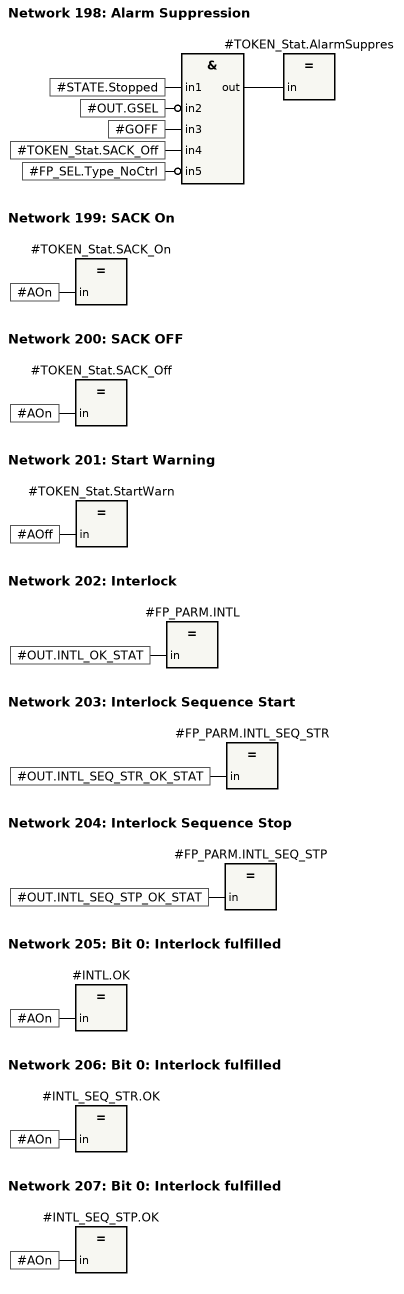
   #TOKEN_Stat.AlarmSuppres := #STATE.Stopped AND NOT #OUT.GSEL AND #GOFF AND #TOKEN_Stat.SACK_Off AND NOT #FP_SEL.Type_NoCtrl;
END_REGION

REGION Network 199: SACK On
   #TOKEN_Stat.SACK_On := #AOn;
END_REGION

REGION Network 200: SACK OFF
   #TOKEN_Stat.SACK_Off := #AOn;
END_REGION

REGION Network 201: Start Warning
   #TOKEN_Stat.StartWarn := #AOff;
END_REGION

REGION Network 202: Interlock
   #FP_PARM.INTL := #OUT.INTL_OK_STAT;
END_REGION

REGION Network 203: Interlock Sequence Start
   #FP_PARM.INTL_SEQ_STR := #OUT.INTL_SEQ_STR_OK_STAT;
END_REGION

REGION Network 204: Interlock Sequence Stop
   #FP_PARM.INTL_SEQ_STP := #OUT.INTL_SEQ_STP_OK_STAT;
END_REGION

REGION Network 205: Bit 0: Interlock fulfilled
   #INTL.OK := #AOn;
END_REGION

REGION Network 206: Bit 0: Interlock fulfilled
   #INTL_SEQ_STR.OK := #AOn;
END_REGION

REGION Network 207: Bit 0: Interlock fulfilled
   #INTL_SEQ_STP.OK := #AOn;
END_REGION

REGION Network 208: Bit 1: Detect first occuring interlock, unit running
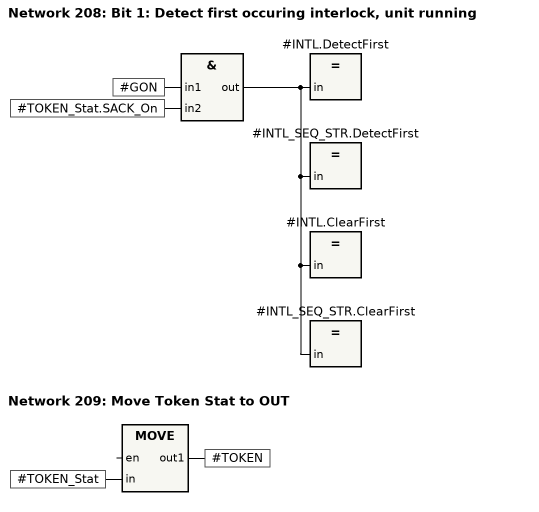
   #INTL.DetectFirst := #GON AND #TOKEN_Stat.SACK_On;
   #INTL_SEQ_STR.DetectFirst := #INTL.DetectFirst;
   #INTL.ClearFirst := #INTL.DetectFirst;
   #INTL_SEQ_STR.ClearFirst := #INTL.DetectFirst;
END_REGION

REGION Network 209: Move Token Stat to OUT
   #TOKEN := #TOKEN_Stat;
END_REGION

REGION Network 210: Write STAT to OUT
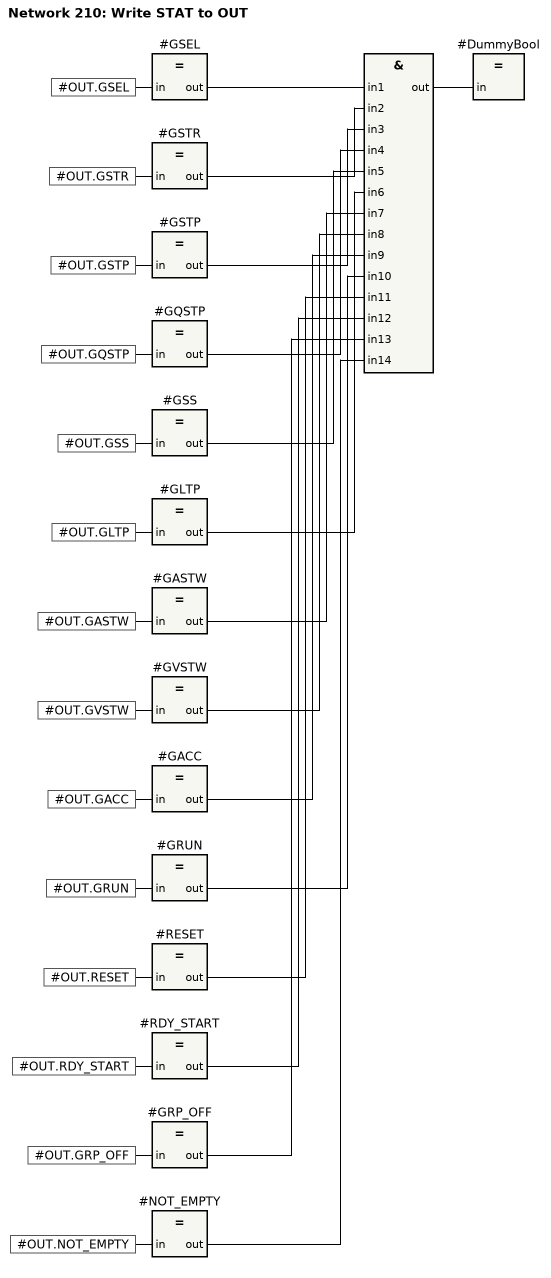
   #GSEL := #OUT.GSEL;
   #GSTR := #OUT.GSTR;
   #GSTP := #OUT.GSTP;
   #GQSTP := #OUT.GQSTP;
   #GSS := #OUT.GSS;
   #GLTP := #OUT.GLTP;
   #GASTW := #OUT.GASTW;
   #GVSTW := #OUT.GVSTW;
   #GACC := #OUT.GACC;
   #GRUN := #OUT.GRUN;
   #RESET := #OUT.RESET;
   #RDY_START := #OUT.RDY_START;
   #GRP_OFF := #OUT.GRP_OFF;
   #NOT_EMPTY := #OUT.NOT_EMPTY;
   #DummyBool := #OUT.GSEL AND #OUT.GSTR AND #OUT.GSTP AND #OUT.GQSTP AND #OUT.GSS AND #OUT.GLTP AND #OUT.GASTW AND #OUT.GVSTW AND #OUT.GACC AND #OUT.GRUN AND #OUT.RESET AND #OUT.RDY_START AND #OUT.GRP_OFF AND #OUT.NOT_EMPTY;
END_REGION
END_FUNCTION_BLOCK

FUNCTION_BLOCK "ACESYS_ALARM"   // FB203, FBD
TITLE = ACESYS V8.0 - Build 004 - Alarm Block
{ S7_Optimized_Access := 'FALSE' }
AUTHOR : FLSmidth
FAMILY : ACESYS
NAME : ALARM
VERSION : 8.0
   VAR_INPUT
      SIG : Bool := TRUE;   // Signal
      PWR : Bool;   // Power Supply
      EN_L : Bool;   // Enable Low Alarm
      EN_H : Bool;   // Enable High Alarm
      AL_SUPR : Bool;   // Alarm Supress by Program
   END_VAR
   VAR_OUTPUT
      OK : Bool;   // Status OK = No Current Alarm
      AL_L : Bool;   // Alarm Low
      AL_H : Bool;   // Alarm High
      WARN_L : Bool;   // Warning Low
      WARN_H : Bool;   // Warning High
      MSW : "ACESYS_HMI_STAT_32T";
   END_VAR
   VAR_IN_OUT
      TOKEN : "ACESYS_TOKEN";
   END_VAR
   VAR
      BlockInfo : Struct
         Ace_Version : Int;   // Acesys Block Version Number
         Ace_BuildNo : Int;   // Acesys Block Build Number
         State_Act : Int;   // Actual State Number
         State_Prev : Int;   // Previous State Number
         DB_Number : Int;   // Block Instance DB Number
      END_STRUCT;
      FP_CMD : Struct   // Faceplate Commands
         Spare_08 : Bool;
         Spare_09 : Bool;
         Spare_10 : Bool;
         Spare_11 : Bool;
         Spare_12 : Bool;
         Spare_13 : Bool;
         Spare_14 : Bool;
         AckAlarm : Bool;
         Spare_00 : Bool;
         Spare_01 : Bool;
         Spare_02 : Bool;
         Spare_03 : Bool;
         Spare_04 : Bool;
         Spare_05 : Bool;
         Spare_06 : Bool;
         Spare_07 : Bool;
      END_STRUCT;
      FP_SEL : Struct
         Force_Low_Alarm : Bool;   // Select Bit
         Force_High_Alarm : Bool;   // Select Bit
         Force_OK : Bool;   // Select Bit
         Force_Low_Warning : Bool;   // Select Bit
         Force_High_Warning : Bool;   // Select Bit
         Keep_Status : Bool;   // Select Bit
         Spare06 : Bool;
         Spare07 : Bool;
         Spare08 : Bool;
         Spare09 : Bool;
         Spare10 : Bool;
         Spare11 : Bool;
         Spare12 : Bool;
         Spare13 : Bool;
         Spare14 : Bool;
         Spare15 : Bool;
      END_STRUCT;
      FP_PARM : Struct
         EnableTime_Low_Pre : Int;
         EnableTime_Low_Acc : Int;
         EnableTime_High_Pre : Int;
         EnableTime_High_Acc : Int;
         WarnDelay_Low_Pre : Int;
         WarnDelay_Low_Acc : Int;
         WarnDelay_High_Pre : Int;
         WarnDelay_High_Acc : Int;
         AlarmDelay_High_Pre : Int;
         AlarmDelay_High_Acc : Int;
         AlarmDelay_Low_Pre : Int;
         AlarmDelay_Low_Acc : Int;
         RepeatTime_Pre : Int;
         RepeatTime_Acc : Int;
         Struct0 : Int;
      END_STRUCT;
      FP_EN : Struct
         ParentSupress : Bool;   // Enable Bit
         ParentSupressUnit : Bool;   // Enable Bit
         Repeat_Alarm : Bool;   // Enable Bit
         Alarm_Low : Bool;   // Enable Bit
         Alarm_High : Bool;   // Enable Bit
         Warning_Low : Bool;   // Enable Bit
         Warning_High : Bool;   // Enable Bit
         Spare07 : Bool;
         Spare08 : Bool;
         Spare09 : Bool;
         Spare10 : Bool;
         Spare11 : Bool;
         Spare12 : Bool;
         Spare13 : Bool;
         Spare14 : Bool;
         Spare15 : Bool;
      END_STRUCT;
      FP_SIM : "ACESYS_SIM_ALARM";
      ONS : Struct
         Sec_Pulse2 : Bool;   // OneShot bit
         Sec_Pulse1 : Bool;   // OneShot bit
         Acknowledge : Bool;   // OneShot bit
         ForceOK : Bool;   // OneShot bit
         ForceLowAlarm : Bool;   // OneShot bit
         ForceHighAlarm : Bool;   // OneShot bit
         SecPulse1 : Bool;
         SecPulse2 : Bool;
         Spare08 : Bool;
         Spare07 : Bool;
         Spare06 : Bool;
         Spare05 : Bool;
         Spare04 : Bool;
         ALARM_AlarmCondition : Bool;
         AL_L_Aux : Bool;
         AL_H_Aux : Bool;
      END_STRUCT;
      EnableTime_Low_Done : Bool;   // Timer Done
      EnableTime_High_Done : Bool;   // Timer Done
      WarnDelay_Low_Done : Bool;   // Timer Done
      WarnDelay_High_Done : Bool;   // Timer Done
      AlarmDelay_Low_Done : Bool;   // Timer Done
      AlarmDelay_High_Done : Bool;   // Timer Done
      RepeatTime_Done : Bool;   // Timer Done
      ALARM_SuppresionActiv : Bool;
      ALARM_AlarmPresent : Bool;
      ALARM_WarnPresent : Bool;
      ALARM_Failure_Ack_Requ : Bool;
      ALARM_Warn_Ack_Required : Bool;
      Keep_L_Alarm : Bool;   // Keep Alarm
      Keep_H_Alarm : Bool;
      Sec_Pulse : Bool;   // Pulse Every Second
      CMD_Acknowledge : Bool;   // Internal Acknowledge
      StatusWork : Int;
      AlarmNo : Int;
      AlarmNo_Old : Int;
      EnableTime_Low_Mem : Int;   // Timer Memory
      EnableTime_High_Mem : Int;   // Timer Memory
      WarnDelay_Low_Mem : Int;   // Timer Memory
      WarnDelay_High_Mem : Int;   // Timer Memory
      AlarmDelay_High_Mem : Int;   // Timer Memory
      AlarmDelay_Low_Mem : Int;   // Timer Memory
      RepeatTime_Mem : Int;   // Timer Memory
      OUT : Struct
         OK : Bool;
         AL_L : Bool;
         AL_H : Bool;
         WARN_L : Bool;
         WARN_H : Bool;
      END_STRUCT;
      MSW_EXT_AlarmFailUnAck : Bool;
      MSW_Status_Trans : Int;
   END_VAR
   VAR_TEMP
      AOn : Bool;   // Always On
      AOff : Bool;   // Always Off
      DummyBool : Bool;
   END_VAR
   VAR_TEMP   // added for the SCL form of the ladder/FBD networks
      _w1 : Bool;
      _w2 : Bool;
      _w3 : Bool;
   END_VAR
BEGIN

REGION Network 1: Always On
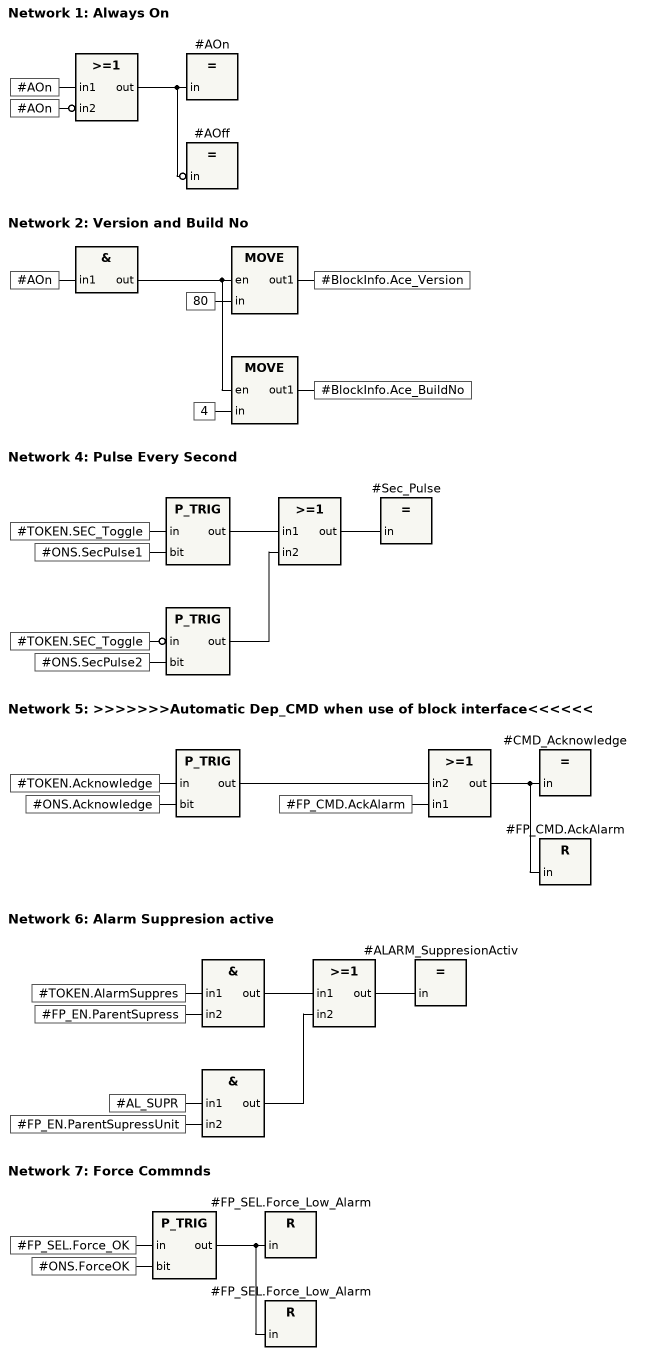
   #AOn := #AOn OR NOT #AOn;
   #AOff := NOT #AOn;
END_REGION

REGION Network 2: Version and Build No
   IF #AOn THEN
       #BlockInfo.Ace_Version := 80;
       #BlockInfo.Ace_BuildNo := 4;
   END_IF;
END_REGION

REGION Network 3 (STL): Instance DB Number to Faceplate
         L     DINO;
         T     #BlockInfo.DB_Number;
END_REGION

REGION Network 4: Pulse Every Second
   #_w1 := #TOKEN.SEC_Toggle AND NOT #ONS.SecPulse1;   // rising edge
   #ONS.SecPulse1 := #TOKEN.SEC_Toggle;
   #_w2 := NOT #TOKEN.SEC_Toggle AND NOT #ONS.SecPulse2;   // rising edge
   #ONS.SecPulse2 := NOT #TOKEN.SEC_Toggle;
   #Sec_Pulse := #_w1 OR #_w2;
END_REGION

REGION Network 5: >>>>>>>Automatic Dep_CMD when use of block interface<<<<<<
   #_w1 := #TOKEN.Acknowledge AND NOT #ONS.Acknowledge;   // rising edge
   #ONS.Acknowledge := #TOKEN.Acknowledge;
   #CMD_Acknowledge := #_w1 OR #FP_CMD.AckAlarm;
   IF #CMD_Acknowledge THEN #FP_CMD.AckAlarm := FALSE; END_IF;
END_REGION

REGION Network 6: Alarm Suppresion active
   #ALARM_SuppresionActiv := (#TOKEN.AlarmSuppres AND #FP_EN.ParentSupress) OR (#AL_SUPR AND #FP_EN.ParentSupressUnit);
END_REGION

REGION Network 7: Force Commnds
   #_w1 := #FP_SEL.Force_OK AND NOT #ONS.ForceOK;   // rising edge
   #ONS.ForceOK := #FP_SEL.Force_OK;
   IF #_w1 THEN
       #FP_SEL.Force_Low_Alarm := FALSE;
       #FP_SEL.Force_Low_Alarm := FALSE;
   END_IF;
END_REGION

REGION Network 8: Select Bit
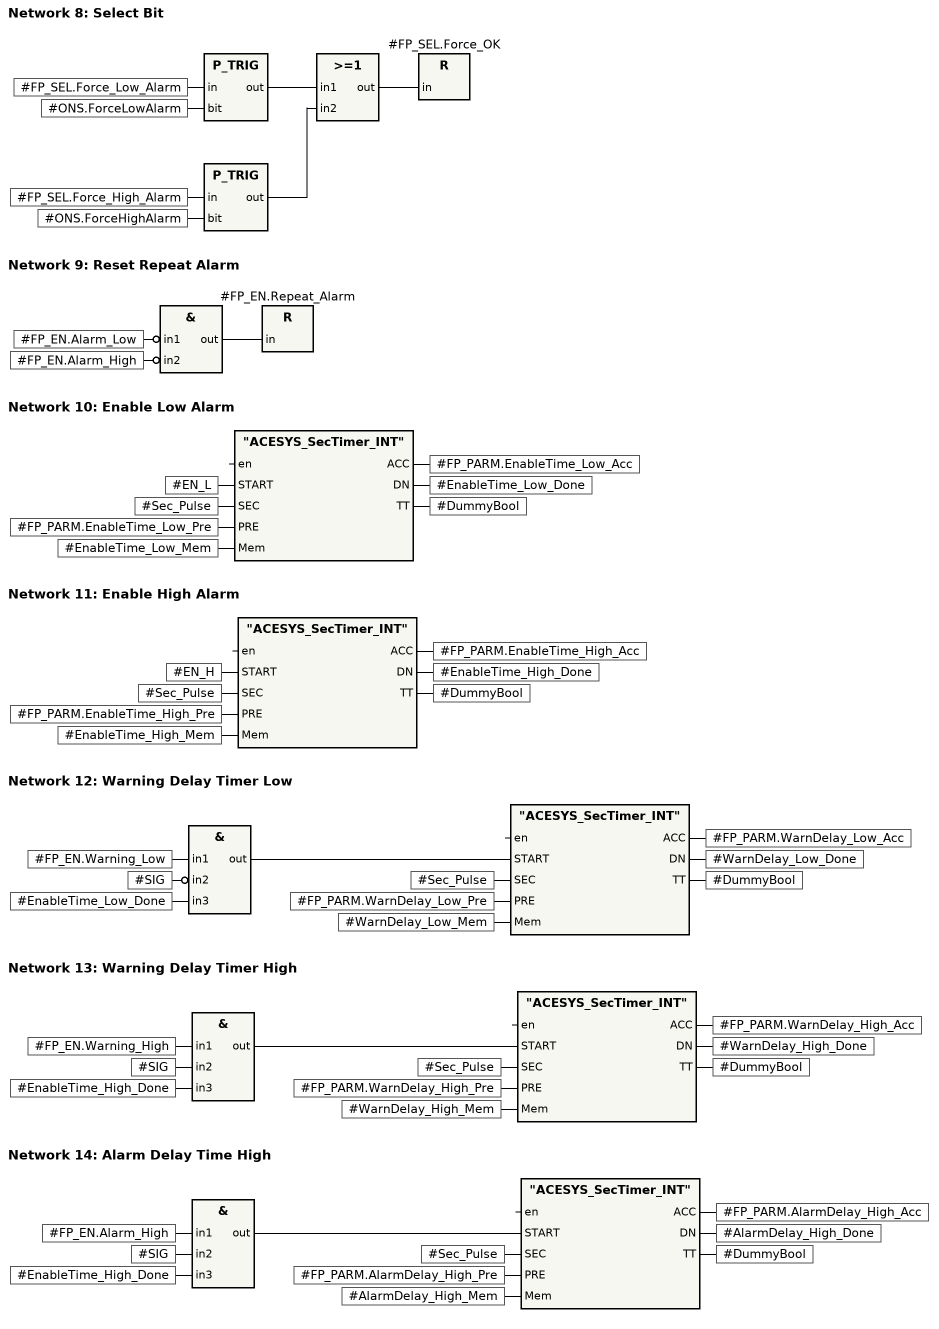
   #_w1 := #FP_SEL.Force_Low_Alarm AND NOT #ONS.ForceLowAlarm;   // rising edge
   #ONS.ForceLowAlarm := #FP_SEL.Force_Low_Alarm;
   #_w2 := #FP_SEL.Force_High_Alarm AND NOT #ONS.ForceHighAlarm;   // rising edge
   #ONS.ForceHighAlarm := #FP_SEL.Force_High_Alarm;
   IF #_w1 OR #_w2 THEN #FP_SEL.Force_OK := FALSE; END_IF;
END_REGION

REGION Network 9: Reset Repeat Alarm
   IF NOT #FP_EN.Alarm_Low AND NOT #FP_EN.Alarm_High THEN #FP_EN.Repeat_Alarm := FALSE; END_IF;
END_REGION

REGION Network 10: Enable Low Alarm
   "ACESYS_SecTimer_INT"(START := #EN_L,
                         SEC := #Sec_Pulse,
                         PRE := #FP_PARM.EnableTime_Low_Pre,
                         Mem := #EnableTime_Low_Mem,
                         ACC => #FP_PARM.EnableTime_Low_Acc,
                         DN => #EnableTime_Low_Done,
                         TT => #DummyBool);
END_REGION

REGION Network 11: Enable High Alarm
   "ACESYS_SecTimer_INT"(START := #EN_H,
                         SEC := #Sec_Pulse,
                         PRE := #FP_PARM.EnableTime_High_Pre,
                         Mem := #EnableTime_High_Mem,
                         ACC => #FP_PARM.EnableTime_High_Acc,
                         DN => #EnableTime_High_Done,
                         TT => #DummyBool);
END_REGION

REGION Network 12: Warning Delay Timer Low
   // Build 002 - 27 March 2019 : EnableTime_Low_Done added
   "ACESYS_SecTimer_INT"(START := #FP_EN.Warning_Low AND NOT #SIG AND #EnableTime_Low_Done,
                         SEC := #Sec_Pulse,
                         PRE := #FP_PARM.WarnDelay_Low_Pre,
                         Mem := #WarnDelay_Low_Mem,
                         ACC => #FP_PARM.WarnDelay_Low_Acc,
                         DN => #WarnDelay_Low_Done,
                         TT => #DummyBool);
END_REGION

REGION Network 13: Warning Delay Timer High
   // Build 002 - 27 March 2019 : EnableTime_High_Done added
   "ACESYS_SecTimer_INT"(START := #FP_EN.Warning_High AND #SIG AND #EnableTime_High_Done,
                         SEC := #Sec_Pulse,
                         PRE := #FP_PARM.WarnDelay_High_Pre,
                         Mem := #WarnDelay_High_Mem,
                         ACC => #FP_PARM.WarnDelay_High_Acc,
                         DN => #WarnDelay_High_Done,
                         TT => #DummyBool);
END_REGION

REGION Network 14: Alarm Delay Time High
   // Build 002 - 27 March 2019 : EnableTime_High_Done added
   "ACESYS_SecTimer_INT"(START := #FP_EN.Alarm_High AND #SIG AND #EnableTime_High_Done,
                         SEC := #Sec_Pulse,
                         PRE := #FP_PARM.AlarmDelay_High_Pre,
                         Mem := #AlarmDelay_High_Mem,
                         ACC => #FP_PARM.AlarmDelay_High_Acc,
                         DN => #AlarmDelay_High_Done,
                         TT => #DummyBool);
END_REGION

REGION Network 15: Alarm Delay Time Low
   // Build 002 - 27 March 2019 : EnableTime_Low_Done added
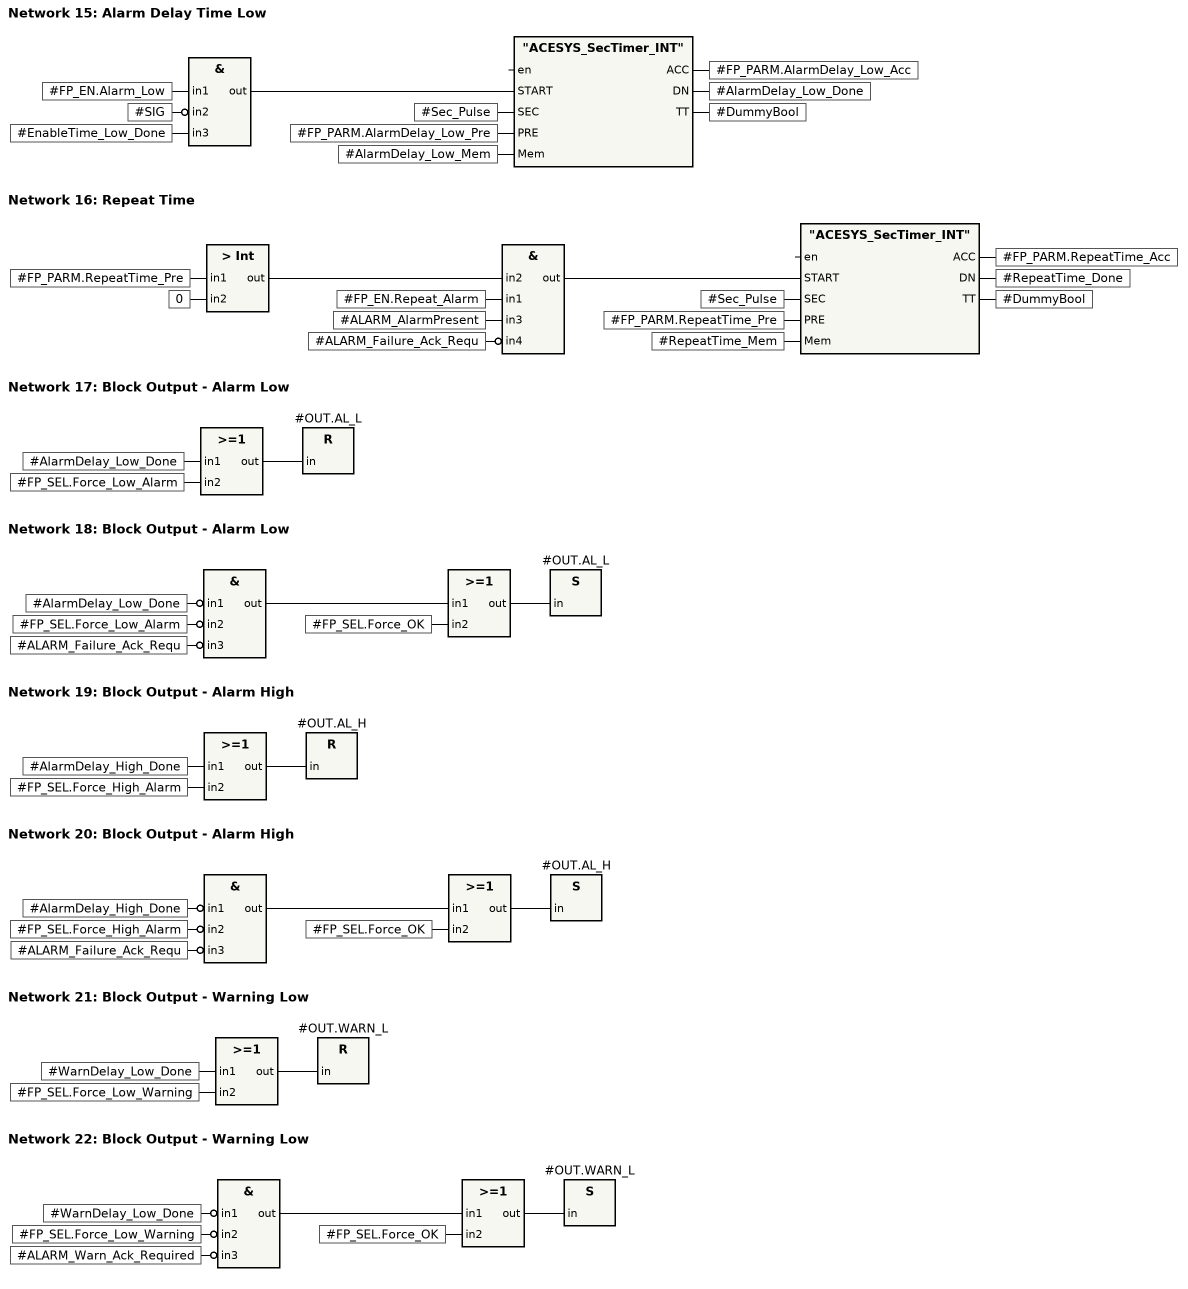
   "ACESYS_SecTimer_INT"(START := #FP_EN.Alarm_Low AND NOT #SIG AND #EnableTime_Low_Done,
                         SEC := #Sec_Pulse,
                         PRE := #FP_PARM.AlarmDelay_Low_Pre,
                         Mem := #AlarmDelay_Low_Mem,
                         ACC => #FP_PARM.AlarmDelay_Low_Acc,
                         DN => #AlarmDelay_Low_Done,
                         TT => #DummyBool);
END_REGION

REGION Network 16: Repeat Time
   "ACESYS_SecTimer_INT"(START := (#FP_PARM.RepeatTime_Pre > 0) AND #FP_EN.Repeat_Alarm AND #ALARM_AlarmPresent AND NOT #ALARM_Failure_Ack_Requ,
                         SEC := #Sec_Pulse,
                         PRE := #FP_PARM.RepeatTime_Pre,
                         Mem := #RepeatTime_Mem,
                         ACC => #FP_PARM.RepeatTime_Acc,
                         DN => #RepeatTime_Done,
                         TT => #DummyBool);
END_REGION

REGION Network 17: Block Output - Alarm Low
   // Build 002 - 27 March 2019 : Deleted EnableTime_Low_Done
   IF #AlarmDelay_Low_Done OR #FP_SEL.Force_Low_Alarm THEN #OUT.AL_L := FALSE; END_IF;
END_REGION

REGION Network 18: Block Output - Alarm Low
   // Build 002 - 26 March 2019 : Deleted EnableTime_Low_Done
   IF (NOT #AlarmDelay_Low_Done AND NOT #FP_SEL.Force_Low_Alarm AND NOT #ALARM_Failure_Ack_Requ) OR #FP_SEL.Force_OK THEN
       #OUT.AL_L := TRUE;
   END_IF;
END_REGION

REGION Network 19: Block Output - Alarm High
   // Build 002 - 26 March 2019 : Deleted EnableTime_High_Done
   IF #AlarmDelay_High_Done OR #FP_SEL.Force_High_Alarm THEN #OUT.AL_H := FALSE; END_IF;
END_REGION

REGION Network 20: Block Output - Alarm High
   // Build 002 - 26 March 2019 : Deleted EnableTime_High_Done
   IF (NOT #AlarmDelay_High_Done AND NOT #FP_SEL.Force_High_Alarm AND NOT #ALARM_Failure_Ack_Requ) OR #FP_SEL.Force_OK THEN
       #OUT.AL_H := TRUE;
   END_IF;
END_REGION

REGION Network 21: Block Output - Warning Low
   // Build 002 - 27 March 2019 : Deleted EnableTime_Low_Done
   IF #WarnDelay_Low_Done OR #FP_SEL.Force_Low_Warning THEN #OUT.WARN_L := FALSE; END_IF;
END_REGION

REGION Network 22: Block Output - Warning Low
   // Build 002 - 27 March 2019 : Deleted EnableTime_Low_Done
   IF (NOT #WarnDelay_Low_Done AND NOT #FP_SEL.Force_Low_Warning AND NOT #ALARM_Warn_Ack_Required) OR #FP_SEL.Force_OK THEN
       #OUT.WARN_L := TRUE;
   END_IF;
END_REGION

REGION Network 23: Block Output - Warning High
   // Build 002 - 27 March 2019 : Deleted EnableTime_High_Done
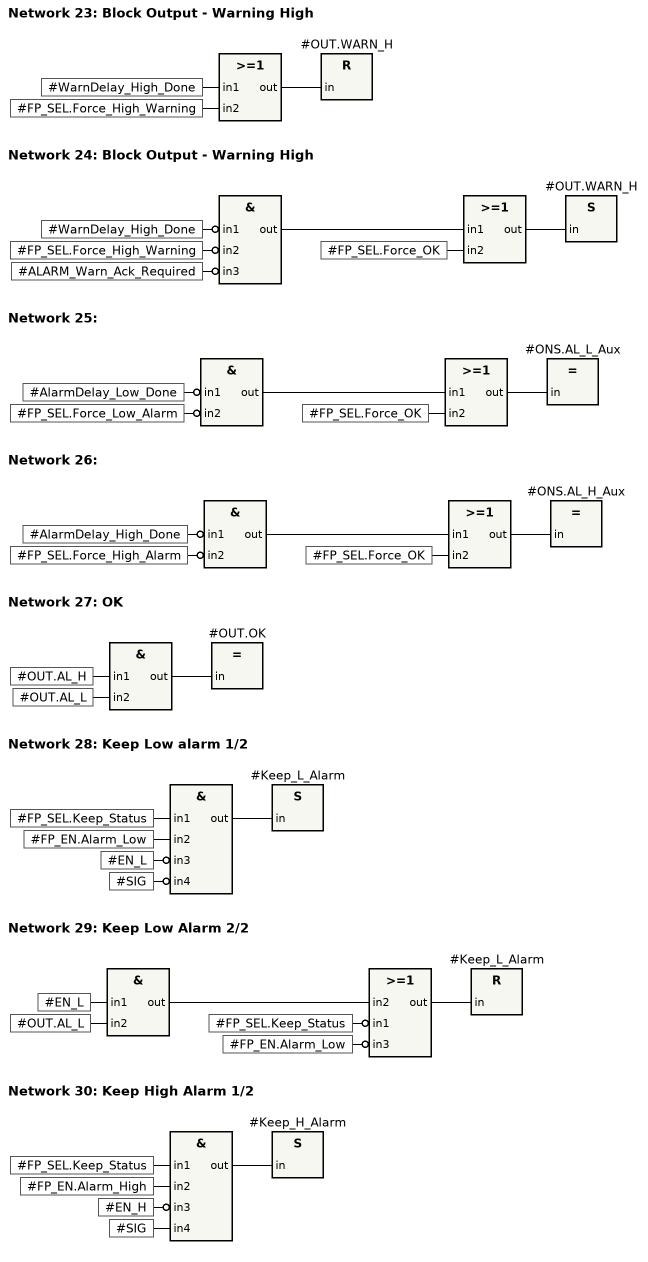
   IF #WarnDelay_High_Done OR #FP_SEL.Force_High_Warning THEN #OUT.WARN_H := FALSE; END_IF;
END_REGION

REGION Network 24: Block Output - Warning High
   // Build 002 - 27 March 2019 : Deleted EnableTime_High_Done
   IF (NOT #WarnDelay_High_Done AND NOT #FP_SEL.Force_High_Warning AND NOT #ALARM_Warn_Ack_Required) OR #FP_SEL.Force_OK THEN
       #OUT.WARN_H := TRUE;
   END_IF;
END_REGION

REGION Network 25
   // Build 002 - 27 March 2019 : New Network
   // Build 003 - 03.July.2019 (EXTBOB): Renamed output bool
   #ONS.AL_L_Aux := (NOT #AlarmDelay_Low_Done AND NOT #FP_SEL.Force_Low_Alarm) OR #FP_SEL.Force_OK;
END_REGION

REGION Network 26
   // Build 003 - 03.July.2019 (EXTBOB): New Network
   #ONS.AL_H_Aux := (NOT #AlarmDelay_High_Done AND NOT #FP_SEL.Force_High_Alarm) OR #FP_SEL.Force_OK;
END_REGION

REGION Network 27: OK
   #OUT.OK := #OUT.AL_H AND #OUT.AL_L;
END_REGION

REGION Network 28: Keep Low alarm 1/2
   IF #FP_SEL.Keep_Status AND #FP_EN.Alarm_Low AND NOT #EN_L AND NOT #SIG THEN #Keep_L_Alarm := TRUE; END_IF;
END_REGION

REGION Network 29: Keep Low Alarm 2/2
   IF (#EN_L AND #OUT.AL_L) OR NOT #FP_SEL.Keep_Status OR NOT #FP_EN.Alarm_Low THEN
       #Keep_L_Alarm := FALSE;
   END_IF;
END_REGION

REGION Network 30: Keep High Alarm 1/2
   IF #FP_SEL.Keep_Status AND #FP_EN.Alarm_High AND NOT #EN_H AND #SIG THEN #Keep_H_Alarm := TRUE; END_IF;
END_REGION

REGION Network 31: Keep High Alarm 2/2
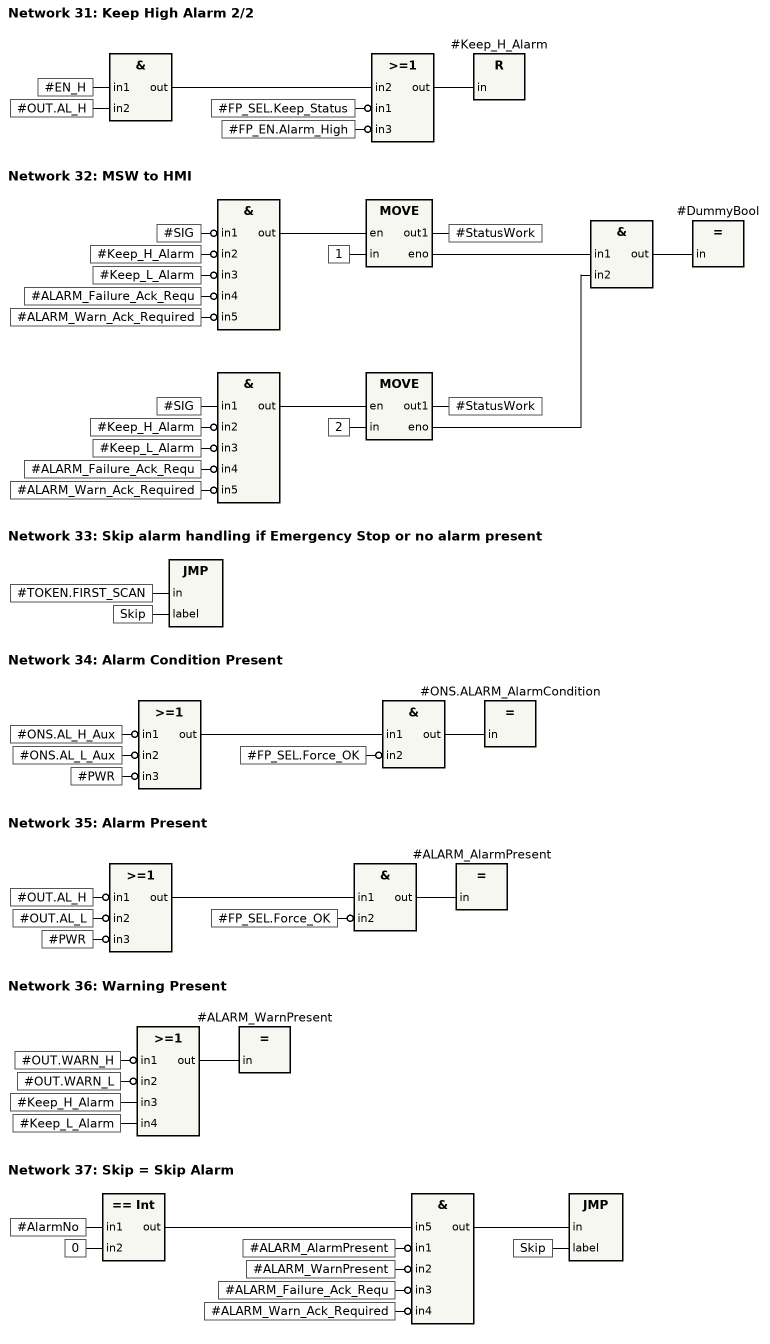
   IF (#EN_H AND #OUT.AL_H) OR NOT #FP_SEL.Keep_Status OR NOT #FP_EN.Alarm_High THEN
       #Keep_H_Alarm := FALSE;
   END_IF;
END_REGION

REGION Network 32: MSW to HMI
   // ENO of a box is taken as its EN; it also drops when the box reports an error
   #_w1 := NOT #SIG AND NOT #Keep_H_Alarm AND NOT #Keep_L_Alarm AND NOT #ALARM_Failure_Ack_Requ AND NOT #ALARM_Warn_Ack_Required;
   IF #_w1 THEN #StatusWork := 1; END_IF;
   #_w2 := #SIG AND NOT #Keep_H_Alarm AND NOT #Keep_L_Alarm AND NOT #ALARM_Failure_Ack_Requ AND NOT #ALARM_Warn_Ack_Required;
   IF #_w2 THEN #StatusWork := 2; END_IF;
   #DummyBool := #_w1 AND #_w2;
END_REGION

REGION Network 33: Skip alarm handling if Emergency Stop or no alarm present
   // Skip = Skip Alarm
   IF #TOKEN.FIRST_SCAN THEN GOTO Skip; END_IF;
END_REGION

REGION Network 34: Alarm Condition Present
   // Build 003 - 03.July.2019 (EXTBOB) - New Network
   #ONS.ALARM_AlarmCondition := (NOT #ONS.AL_H_Aux OR NOT #ONS.AL_L_Aux OR NOT #PWR) AND NOT #FP_SEL.Force_OK;
END_REGION

REGION Network 35: Alarm Present
   #ALARM_AlarmPresent := (NOT #OUT.AL_H OR NOT #OUT.AL_L OR NOT #PWR) AND NOT #FP_SEL.Force_OK;
END_REGION

REGION Network 36: Warning Present
   #ALARM_WarnPresent := NOT #OUT.WARN_H OR NOT #OUT.WARN_L OR #Keep_H_Alarm OR #Keep_L_Alarm;
END_REGION

REGION Network 37: Skip = Skip Alarm
   IF (#AlarmNo = 0) AND NOT #ALARM_AlarmPresent AND NOT #ALARM_WarnPresent AND NOT #ALARM_Failure_Ack_Requ AND NOT #ALARM_Warn_Ack_Required THEN
       GOTO Skip;
   END_IF;
END_REGION

REGION Network 38: Clr = Clear Alarm
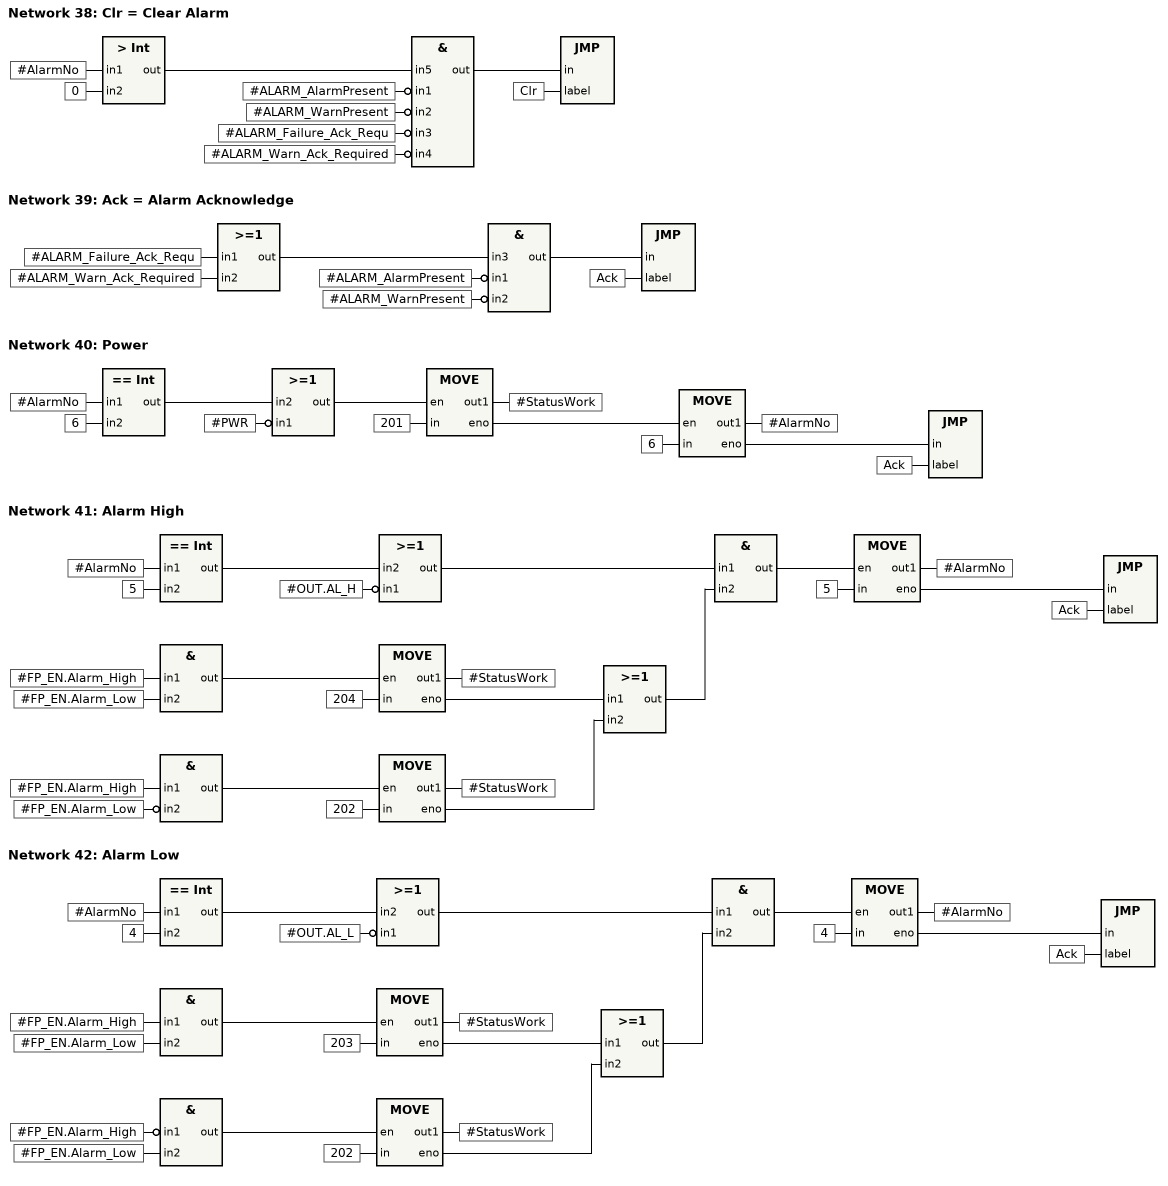
   IF (#AlarmNo > 0) AND NOT #ALARM_AlarmPresent AND NOT #ALARM_WarnPresent AND NOT #ALARM_Failure_Ack_Requ AND NOT #ALARM_Warn_Ack_Required THEN
       GOTO Clr;
   END_IF;
END_REGION

REGION Network 39: Ack = Alarm Acknowledge
   IF (#ALARM_Failure_Ack_Requ OR #ALARM_Warn_Ack_Required) AND NOT #ALARM_AlarmPresent AND NOT #ALARM_WarnPresent THEN
       GOTO Ack;
   END_IF;
END_REGION

REGION Network 40: Power
   // ENO of a box is taken as its EN; it also drops when the box reports an error
   #_w1 := (#AlarmNo = 6) OR NOT #PWR;
   IF #_w1 THEN
       #StatusWork := 201;
       #AlarmNo := 6;
       GOTO Ack;
   END_IF;
END_REGION

REGION Network 41: Alarm High
   // ENO of a box is taken as its EN; it also drops when the box reports an error
   #_w1 := #FP_EN.Alarm_High AND #FP_EN.Alarm_Low;
   IF #_w1 THEN #StatusWork := 204; END_IF;
   #_w2 := #FP_EN.Alarm_High AND NOT #FP_EN.Alarm_Low;
   IF #_w2 THEN #StatusWork := 202; END_IF;
   #_w3 := ((#AlarmNo = 5) OR NOT #OUT.AL_H) AND (#_w1 OR #_w2);
   IF #_w3 THEN
       #AlarmNo := 5;
       GOTO Ack;
   END_IF;
END_REGION

REGION Network 42: Alarm Low
   // ENO of a box is taken as its EN; it also drops when the box reports an error
   #_w1 := #FP_EN.Alarm_High AND #FP_EN.Alarm_Low;
   IF #_w1 THEN #StatusWork := 203; END_IF;
   #_w2 := NOT #FP_EN.Alarm_High AND #FP_EN.Alarm_Low;
   IF #_w2 THEN #StatusWork := 202; END_IF;
   #_w3 := ((#AlarmNo = 4) OR NOT #OUT.AL_L) AND (#_w1 OR #_w2);
   IF #_w3 THEN
       #AlarmNo := 4;
       GOTO Ack;
   END_IF;
END_REGION

REGION Network 43: Warning High
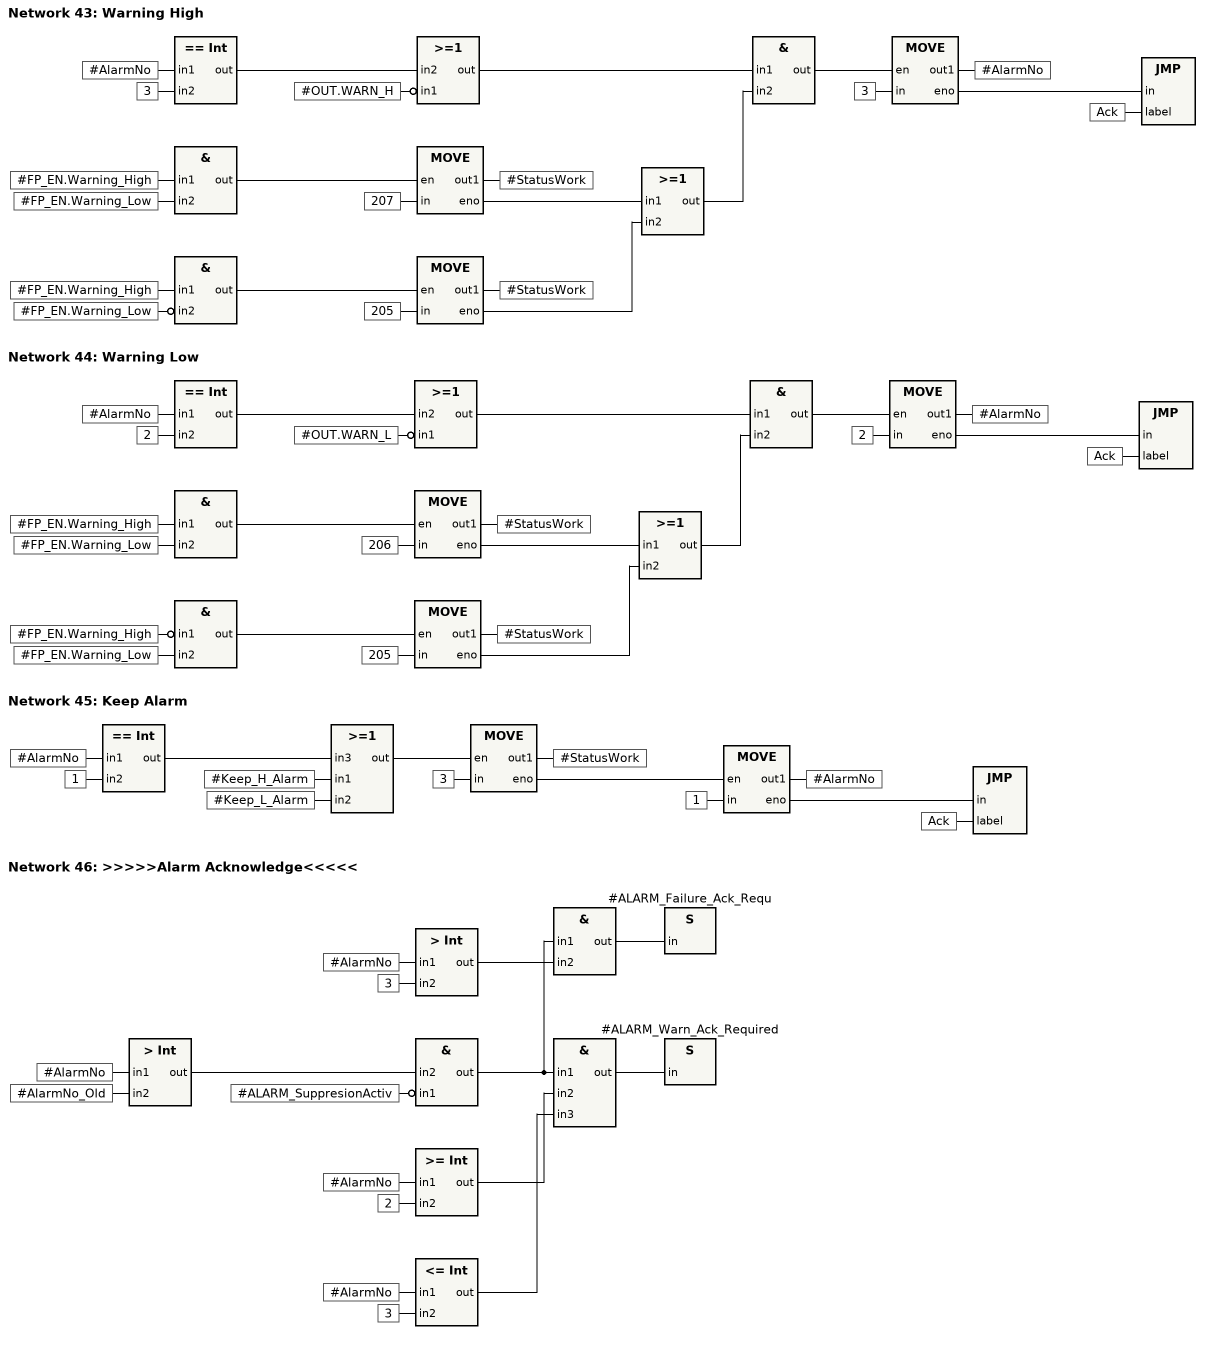
   // ENO of a box is taken as its EN; it also drops when the box reports an error
   #_w1 := #FP_EN.Warning_High AND #FP_EN.Warning_Low;
   IF #_w1 THEN #StatusWork := 207; END_IF;
   #_w2 := #FP_EN.Warning_High AND NOT #FP_EN.Warning_Low;
   IF #_w2 THEN #StatusWork := 205; END_IF;
   #_w3 := ((#AlarmNo = 3) OR NOT #OUT.WARN_H) AND (#_w1 OR #_w2);
   IF #_w3 THEN
       #AlarmNo := 3;
       GOTO Ack;
   END_IF;
END_REGION

REGION Network 44: Warning Low
   // ENO of a box is taken as its EN; it also drops when the box reports an error
   #_w1 := #FP_EN.Warning_High AND #FP_EN.Warning_Low;
   IF #_w1 THEN #StatusWork := 206; END_IF;
   #_w2 := NOT #FP_EN.Warning_High AND #FP_EN.Warning_Low;
   IF #_w2 THEN #StatusWork := 205; END_IF;
   #_w3 := ((#AlarmNo = 2) OR NOT #OUT.WARN_L) AND (#_w1 OR #_w2);
   IF #_w3 THEN
       #AlarmNo := 2;
       GOTO Ack;
   END_IF;
END_REGION

REGION Network 45: Keep Alarm
   // Build 004 - 15.Sept.2020 (MIA-US): AlarmNo comparison corrected (was 0 instead of 1)
   // ENO of a box is taken as its EN; it also drops when the box reports an error
   #_w1 := (#AlarmNo = 1) OR #Keep_H_Alarm OR #Keep_L_Alarm;
   IF #_w1 THEN
       #StatusWork := 3;
       #AlarmNo := 1;
       GOTO Ack;
   END_IF;
END_REGION

REGION Network 46: >>>>>Alarm Acknowledge<<<<<
   Ack:
   #_w1 := (#AlarmNo > #AlarmNo_Old) AND NOT #ALARM_SuppresionActiv;
   IF #_w1 AND (#AlarmNo > 3) THEN #ALARM_Failure_Ack_Requ := TRUE; END_IF;
   IF #_w1 AND (#AlarmNo >= 2) AND (#AlarmNo <= 3) THEN #ALARM_Warn_Ack_Required := TRUE; END_IF;
END_REGION

REGION Network 47
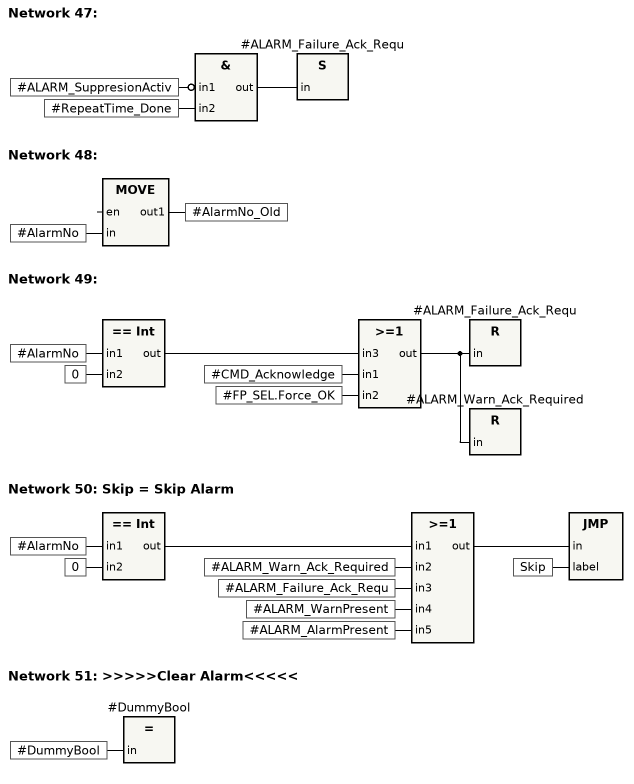
   IF NOT #ALARM_SuppresionActiv AND #RepeatTime_Done THEN #ALARM_Failure_Ack_Requ := TRUE; END_IF;
END_REGION

REGION Network 48
   #AlarmNo_Old := #AlarmNo;
END_REGION

REGION Network 49
   IF (#AlarmNo = 0) OR #CMD_Acknowledge OR #FP_SEL.Force_OK THEN
       #ALARM_Failure_Ack_Requ := FALSE;
       #ALARM_Warn_Ack_Required := FALSE;
   END_IF;
END_REGION

REGION Network 50: Skip = Skip Alarm
   // Build 002 - 27 March 2019: Enable Logic condition alarm no logging is fixed. Alarm_WarnPresent & Alarm_AlarmPresent added to OR gate
   IF (#AlarmNo = 0) OR #ALARM_Warn_Ack_Required OR #ALARM_Failure_Ack_Requ OR #ALARM_WarnPresent OR #ALARM_AlarmPresent THEN
       GOTO Skip;
   END_IF;
END_REGION

REGION Network 51: >>>>>Clear Alarm<<<<<
   Clr:
   #DummyBool := #DummyBool;
END_REGION

REGION Network 52
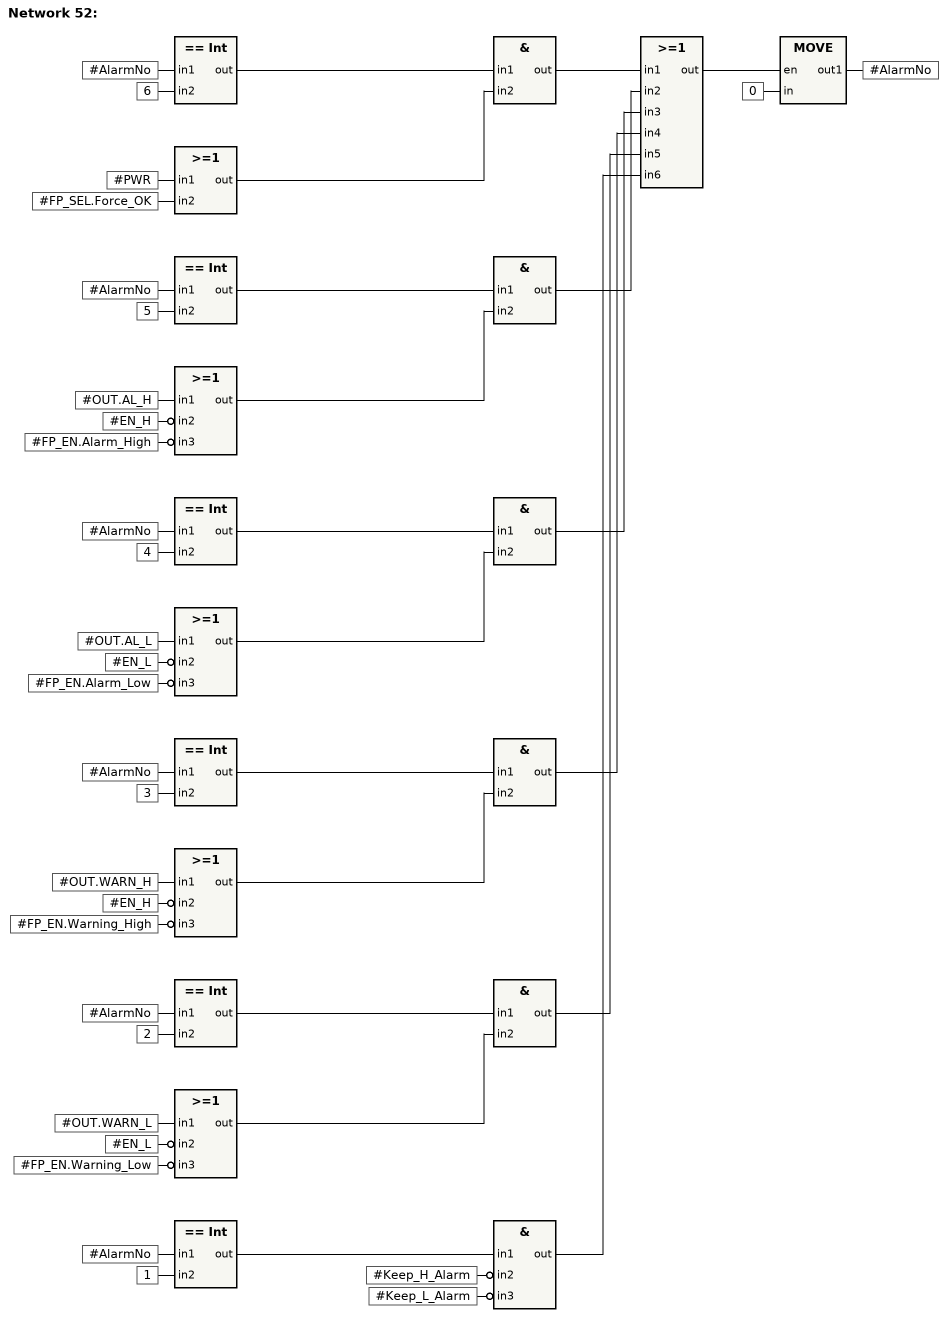
   IF ((#AlarmNo = 6) AND (#PWR OR #FP_SEL.Force_OK)) OR ((#AlarmNo = 5) AND (#OUT.AL_H OR NOT #EN_H OR NOT #FP_EN.Alarm_High)) OR ((#AlarmNo = 4) AND (#OUT.AL_L OR NOT #EN_L OR NOT #FP_EN.Alarm_Low)) OR ((#AlarmNo = 3) AND (#OUT.WARN_H OR NOT #EN_H OR NOT #FP_EN.Warning_High)) OR ((#AlarmNo = 2) AND (#OUT.WARN_L OR NOT #EN_L OR NOT #FP_EN.Warning_Low)) OR ((#AlarmNo = 1) AND NOT #Keep_H_Alarm AND NOT #Keep_L_Alarm) THEN
       #AlarmNo := 0;
   END_IF;
END_REGION

REGION Network 53
   // Build 002 - 27 March 2019 : Replaced ALARM_AlarmPresent with ALARM_AlarmCondition
   // Build 003 - 03.July.2019 (EXTBOB): Typo corrected
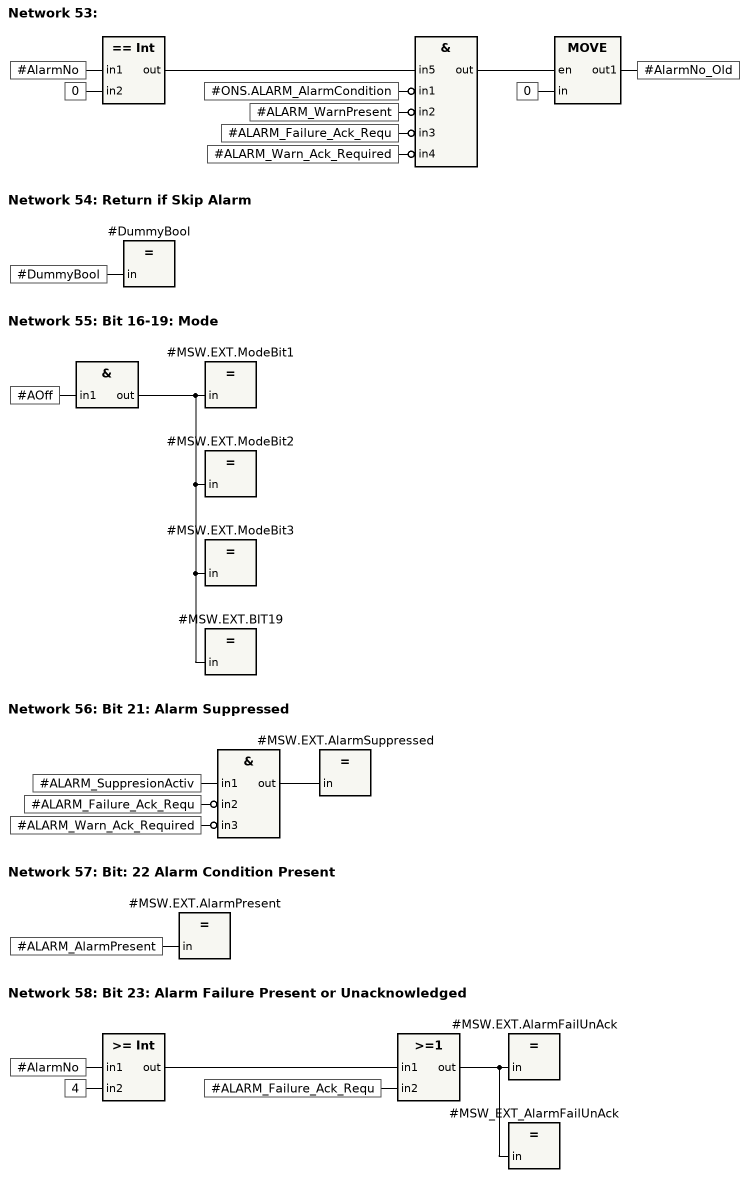
   IF (#AlarmNo = 0) AND NOT #ONS.ALARM_AlarmCondition AND NOT #ALARM_WarnPresent AND NOT #ALARM_Failure_Ack_Requ AND NOT #ALARM_Warn_Ack_Required THEN
       #AlarmNo_Old := 0;
   END_IF;
END_REGION

REGION Network 54: Return if Skip Alarm
   Skip:
   #DummyBool := #DummyBool;
END_REGION

REGION Network 55: Bit 16-19: Mode
   // 0 = Auto
   // 1= Single Start
   // 2 = Manual
   // 3= Local
   // 4= Test Mode
   #MSW.EXT.ModeBit1 := #AOff;
   #MSW.EXT.ModeBit2 := #AOff;
   #MSW.EXT.ModeBit3 := #AOff;
   #MSW.EXT.BIT19 := #AOff;
END_REGION

REGION Network 56: Bit 21: Alarm Suppressed
   #MSW.EXT.AlarmSuppressed := #ALARM_SuppresionActiv AND NOT #ALARM_Failure_Ack_Requ AND NOT #ALARM_Warn_Ack_Required;
END_REGION

REGION Network 57: Bit: 22 Alarm Condition Present
   #MSW.EXT.AlarmPresent := #ALARM_AlarmPresent;
END_REGION

REGION Network 58: Bit 23: Alarm Failure Present or Unacknowledged
   #MSW.EXT.AlarmFailUnAck := (#AlarmNo >= 4) OR #ALARM_Failure_Ack_Requ;
   #MSW_EXT_AlarmFailUnAck := #MSW.EXT.AlarmFailUnAck;
END_REGION

REGION Network 59: Bit 24: Alarm Warning Present Or Unacknowledged
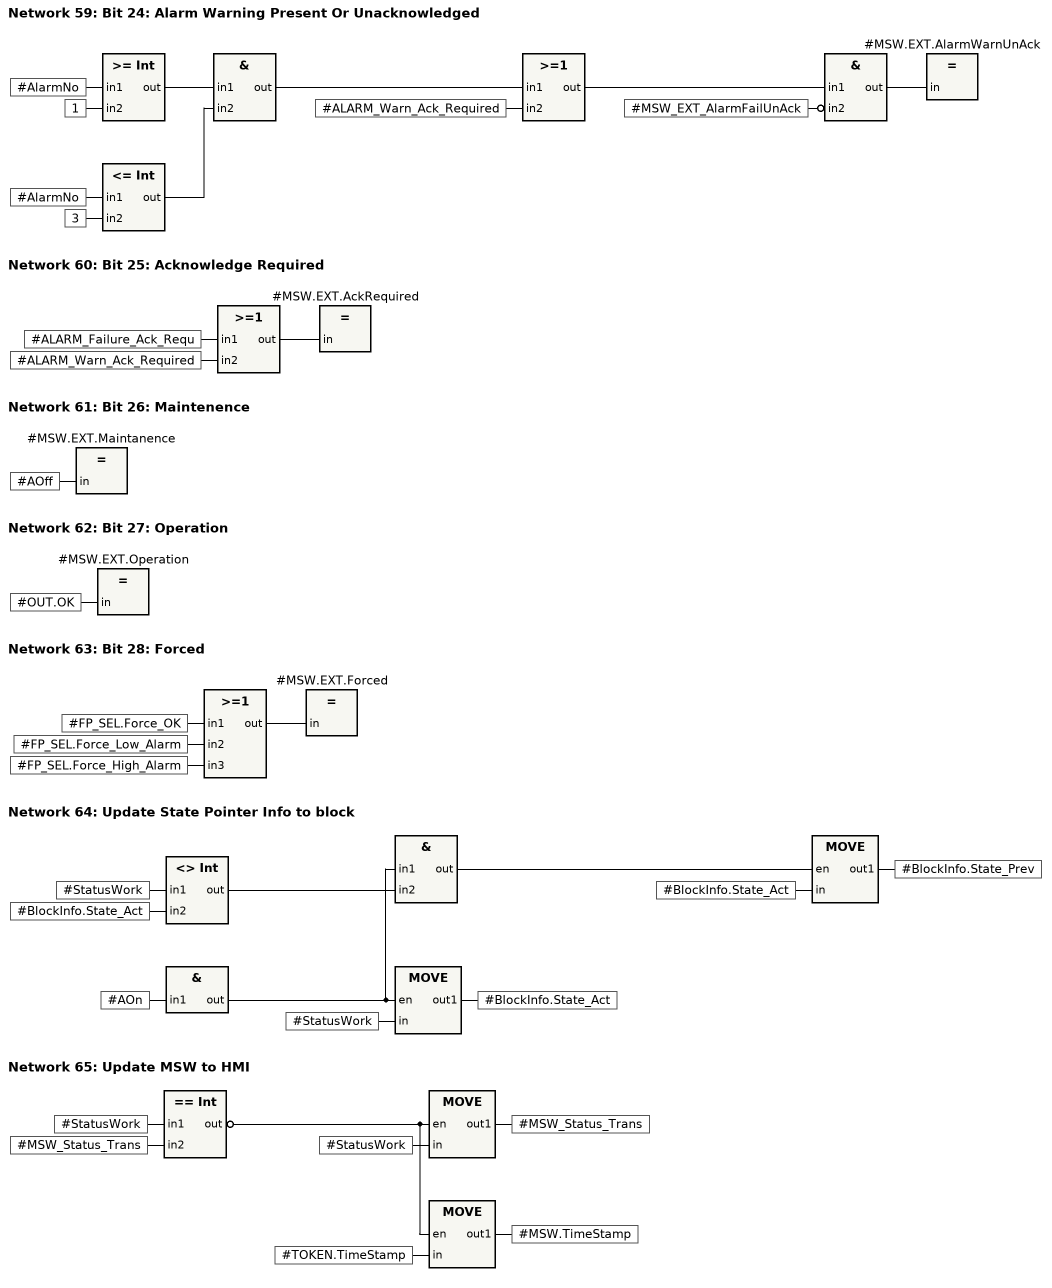
   #MSW.EXT.AlarmWarnUnAck := (((#AlarmNo >= 1) AND (#AlarmNo <= 3)) OR #ALARM_Warn_Ack_Required) AND NOT #MSW_EXT_AlarmFailUnAck;
END_REGION

REGION Network 60: Bit 25: Acknowledge Required
   #MSW.EXT.AckRequired := #ALARM_Failure_Ack_Requ OR #ALARM_Warn_Ack_Required;
END_REGION

REGION Network 61: Bit 26: Maintenence
   #MSW.EXT.Maintanence := #AOff;
END_REGION

REGION Network 62: Bit 27: Operation
   #MSW.EXT.Operation := #OUT.OK;
END_REGION

REGION Network 63: Bit 28: Forced
   #MSW.EXT.Forced := #FP_SEL.Force_OK OR #FP_SEL.Force_Low_Alarm OR #FP_SEL.Force_High_Alarm;
END_REGION

REGION Network 64: Update State Pointer Info to block
   IF #AOn AND (#StatusWork <> #BlockInfo.State_Act) THEN
       #BlockInfo.State_Prev := #BlockInfo.State_Act;
   END_IF;
   IF #AOn THEN #BlockInfo.State_Act := #StatusWork; END_IF;
END_REGION

REGION Network 65: Update MSW to HMI
   #_w1 := NOT (#StatusWork = #MSW_Status_Trans);
   IF #_w1 THEN
       #MSW_Status_Trans := #StatusWork;
       #MSW.TimeStamp := #TOKEN.TimeStamp;
   END_IF;
END_REGION

REGION Network 66: MSW Transfer to Actual
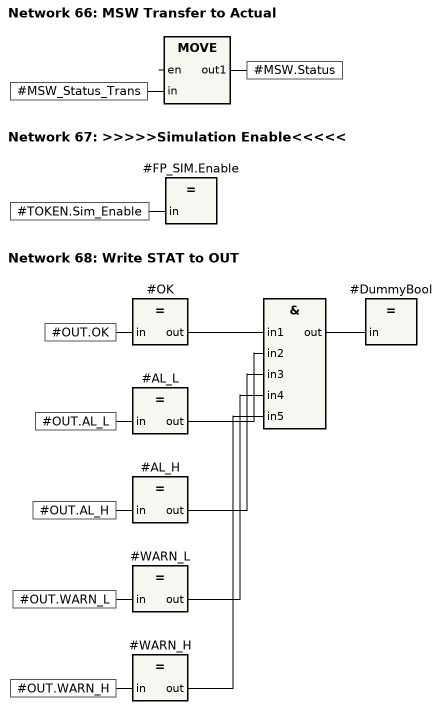
   #MSW.Status := #MSW_Status_Trans;
END_REGION

REGION Network 67: >>>>>Simulation Enable<<<<<
   #FP_SIM.Enable := #TOKEN.Sim_Enable;
END_REGION

REGION Network 68: Write STAT to OUT
   #OK := #OUT.OK;
   #AL_L := #OUT.AL_L;
   #AL_H := #OUT.AL_H;
   #WARN_L := #OUT.WARN_L;
   #WARN_H := #OUT.WARN_H;
   #DummyBool := #OUT.OK AND #OUT.AL_L AND #OUT.AL_H AND #OUT.WARN_L AND #OUT.WARN_H;
END_REGION
END_FUNCTION_BLOCK

FUNCTION_BLOCK "ACESYS_ANALOG"   // FB204, FBD
TITLE = ACESYS V8.0 - Build 001 - Analog Block / ACESYS V8.0 - Build 003 - Analog Block
{ S7_Optimized_Access := 'FALSE' }
AUTHOR : FLSmidth
FAMILY : ACESYS
NAME : ANALOG
VERSION : 8.0
   VAR_INPUT
      SIG_TYPE : Int;   // Signal Type: 0= Normalized 0-100, 1= Eng. Units, 2 = PA Version 3
      IN : Real;   // Process Input Value
      FI_BUS : Byte;   // Field Bus Status
      U_RANGE : Bool;   // Under Range Fault (1 = o
      O_RANGE : Bool;   // Over Range Fault ( 1 = ok)
      SIG_FAULT : Bool;   // Signal Fault (1 = ok)
      EnConfig : Bool;   // Allow change of range and alarm limits from ECS
      AEN : Bool;   // Enable Alarm
      AL_SUPR : Bool;   // Alarm Suppres by Program
   END_VAR
   VAR_OUTPUT
      PV_NORM : Real;   // Process Value normalized 0-100%
      PV_SCAL : Real;   // Process Value Eng. Units
      AL_H3 : Bool;   // Alarm H3
      AL_H2 : Bool;   // Alarm H2
      AL_H1 : Bool;   // Alarm H1
      AL_L1 : Bool;   // Alarm L1
      AL_L2 : Bool;   // Alarm L2
      AL_L3 : Bool;   // Alarm L3
      SIG_OK : Bool;   // Signal Valid
      LIM_H2 : Bool;   // Auxiliary Limit High 2
      LIM_H1 : Bool;   // Auxiliary Limit High 1
      LIM_L1 : Bool;   // Auxiliary Limit Low 1
      LIM_L2 : Bool;   // Auxiliary Limit Low 2
      GR_P : Bool;   // Gradient Positive Limit
      GR_N : Bool;   // Gradient Negative Limit
      MSW : "ACESYS_HMI_STAT_ANALOG";
   END_VAR
   VAR_IN_OUT
      TOKEN : "ACESYS_TOKEN";
   END_VAR
   VAR
      BlockInfo : Struct
         Ace_Version : Int;   // Acesys Block Version Number
         Ace_BuildNo : Int;   // Acesys Block Build Number
         DB_Number : Int;   // Block Instance DB Number
      END_STRUCT;
      FP_CMD : Struct   // Faceplate Commands
         Spare_08 : Bool;
         Spare_09 : Bool;
         Spare_10 : Bool;
         Spare_11 : Bool;
         Spare_12 : Bool;
         Spare_13 : Bool;
         Spare_14 : Bool;
         AckAlarm : Bool;
         Spare_00 : Bool;
         Spare_01 : Bool;
         Spare_02 : Bool;
         Spare_03 : Bool;
         Spare_04 : Bool;
         Spare_05 : Bool;
         Spare_06 : Bool;
         Spare_07 : Bool;
      END_STRUCT;
      FP_EN : Struct
         Square : Bool;   // Enable Bit
         SquareRoot : Bool;   // Enable Bit
         ParentSupress : Bool;   // Enable Bit
         ParentSupressUnit : Bool;   // Enable Bit
         Force : Bool;   // Enable Bit
         Damping : Bool;   // Enable Bit
         Gradient_Pos : Bool;   // Enable Bit
         Gradient_Neg : Bool;   // Enable Bit
         Hysteresis : Bool;   // Enable Bit
         Alarm_H3 : Bool;   // Enable Bit
         Alarm_H2 : Bool;   // Enable Bit
         Alarm_H1 : Bool;   // Enable Bit
         Alarm_L1 : Bool;   // Enable Bit
         Alarm_L2 : Bool;   // Enable Bit
         Alarm_L3 : Bool;   // Enable Bit
         AlarmDelay_H3 : Bool;   // Enable Bit
         AlarmDelay_H2 : Bool;   // Enable Bit
         AlarmDelay_H1 : Bool;   // Enable Bit
         AlarmDelay_L1 : Bool;   // Enable Bit
         AlarmDelay_L2 : Bool;   // Enable Bit
         AlarmDelay_L3 : Bool;   // Enable Bit
         ROC_Warn : Bool;   // Enable Bit
         U_Range_Warn : Bool := TRUE;   // Enable Bit
         O_Range_Warn : Bool := TRUE;   // Enable Bit
      END_STRUCT;
      FP_PARM : Struct
         DampingTime : Int;
         Force_Value : Real;
         Scale_Min : Real;
         Scale_Max : Real := 100.0;
         Gradient : Real;
         Grad_Pos : Real := 1.0;   // Gradient Positiv Limit
         Grad_Neg : Real := 1.0;   // Gradient Negativ Limit
         Grad_X : Real := 1.0;
         Gradient_Time_Pre : Int := 60;   // Timer SP
         Gradient_Time_ACC : Int := 60;   // Timer PV
         Alarm_Hyst : Real;   // Hysteresis
         AlarmLimit_H3 : Real;
         AlarmLimit_H2 : Real;
         AlarmLimit_H1 : Real;
         AlarmLimit_L1 : Real;
         AlarmLimit_L2 : Real;
         AlarmLimit_L3 : Real;
         AlarmDelay_H3_Pre : Int;   // Timer SP
         AlarmDelay_H3_Acc : Int;   // Timer PV
         AlarmDelay_H2_Pre : Int;   // Timer SP
         AlarmDelay_H2_Acc : Int;   // Timer PV
         AlarmDelay_H1_Pre : Int;   // Timer SP
         AlarmDelay_H1_Acc : Int;   // Timer PV
         AlarmDelay_L1_Pre : Int;   // Timer SP
         AlarmDelay_L1_Acc : Int;   // Timer PV
         AlarmDelay_L2_Pre : Int;   // Timer SP
         AlarmDelay_L2_Acc : Int;   // Timer PV
         AlarmDelay_L3_Pre : Int;   // Timer SP
         AlarmDelay_L3_Acc : Int;   // Timer PV
         OpenLoopDelay_Pre : Int;   // Timer SP
         OpenLoopDelay_Acc : Int;   // Timer PV
         OverRangeDelay_Pre : Int;   // Timer SP
         OverRangeDelay_Acc : Int;   // Timer PV
         AuxLimit_H2_Value : Real;
         AuxLimit_H1_Value : Real;
         AuxLimit_L2_Value : Real;
         AuxLimit_L1_Value : Real;
      END_STRUCT;
      FP_SIM : "ACESYS_SIM_ANALOG";
      ONS : Struct
         SecPulse1 : Bool;   // Oneshot Bit
         SecPulse2 : Bool;   // Oneshot Bit
         Acknowledge : Bool;   // Oneshot Bit
         DampingOn : Bool;   // OneShot Bit
         TrigSquare : Bool;   // OneShot Bit
         TrigSquareRoot : Bool;   // OneShot Bit
         GradPosCond : Bool;   // OneShot Bit
         GradNegCond : Bool;   // OneShot Bit
      END_STRUCT;
      FIBUS_SubStatus : Byte;
      FIBUS_Quality : Byte;
      FIBUS_Limit : Byte;
      Result_Smooth : Real;
      Result_Sqrt : Real;
      Result_Square : Real;
      DampXA : Real;
      DampXE : Real;
      DampXEA : Real;
      DampTA : Real;
      DampTG : Real;
      Sec_Pulse : Bool;   // Pulse Every Second
      CMD_Acknowledge : Bool;   // Internal Acknowledge
      ALARM_SuppresionActiv : Bool;
      ALARM_AlarmPresent : Bool;
      ALARM_Failure_Ack_Requ : Bool;
      ALARM_Warn_Ack_Requ : Bool;
      ALARM_WarnPresent : Bool;
      Trig_OpenLoop : Bool;
      Trig_OverRange : Bool;
      Trig_SigFault : Bool;
      AlarmCond_H1 : Bool;
      AlarmCond_H2 : Bool;
      AlarmCond_H3 : Bool;
      AlarmCond_L1 : Bool;
      AlarmCond_L2 : Bool;
      AlarmCond_L3 : Bool;
      AlarmCond_ROC : Bool;   // Rate Of Change
      AlarmDelay_H3_Done : Bool;   // Timer Done
      AlarmDelay_H2_Done : Bool;   // Timer Done
      AlarmDelay_H1_Done : Bool;   // Timer Done
      AlarmDelay_L3_Done : Bool;   // Timer Done
      AlarmDelay_L2_Done : Bool;   // Timer Done
      AlarmDelay_L1_Done : Bool;   // Timer Done
      AlarmDelay_OpenLoop_Done : Bool;   // Timer Done
      AlarmDelay_OverRange_Don : Bool;   // Timer Done
      Gradient_Done : Bool;   // Timer Done
      Gradient_NegAlarm_Cond : Bool;
      Gradient_PosAlarm_Cond : Bool;
      AlarmNo : Int;   // Alarm Number
      AlarmNo_Old : Int;
      StatusWork : Int;
      AlarmDelay_H3_Mem : Int;   // Timer Memory
      AlarmDelay_H2_Mem : Int;   // Timer Memory
      AlarmDelay_H1_Mem : Int;   // Timer Memory
      AlarmDelay_L1_Mem : Int;   // Timer Memory
      AlarmDelay_L2_Mem : Int;   // Timer Memory
      AlarmDelay_L3_Mem : Int;   // Timer Memory
      GradientTime_Mem : Int;   // Timer Memory
      AlarmDelay_OpenLoop_Mem : Int;   // Timer Memory
      AlarmDelay_OverRange_Mem : Int;   // Timer Memory
      ScaledValue : Real;
      Grad_Delta : Real;
      Grad_OldValue : Real;
      HystCalc : Real;
      OUT : Struct
         PV_NORM : Real;
         PV_SCAL : Real;
         AL_H3 : Bool;
         AL_H2 : Bool;
         AL_H1 : Bool;
         AL_L1 : Bool;
         AL_L2 : Bool;
         AL_L3 : Bool;
         SIG_OK : Bool;
         LIM_H2 : Bool;
         LIM_H1 : Bool;
         LIM_L1 : Bool;
         LIM_L2 : Bool;
         GR_P : Bool;
         GR_N : Bool;
      END_STRUCT;
      MSW_EXT_AlarmFailUnAck : Bool;
      MSW_Status_Trans : Int;
   END_VAR
   VAR_TEMP
      FI_BUS_0 : Bool;   // Raw Field Bus status bit 0
      FI_BUS_1 : Bool;   // Raw Field Bus status bit 1
      FI_BUS_2 : Bool;   // Raw Field Bus status bit 2
      FI_BUS_3 : Bool;   // Raw Field Bus status bit 3
      FI_BUS_4 : Bool;   // Raw Field Bus status bit 4
      FI_BUS_5 : Bool;   // Raw Field Bus status bit 5
      FI_BUS_6 : Bool;   // Raw Field Bus status bit 6
      AOn : Bool;   // Always On
      AOff : Bool;   // Always Off
      DummyBool : Bool;
      AlarmCond_BadNonSpec : Bool;
      FI_BUS_7 : Bool;   // Raw Field Bus status bit 7
      AlarmCond_BadConfError : Bool;
      AlarmCond_BadNotConnect : Bool;
      AlarmCond_BadDevFail : Bool;
      AlarmCond_BadSensFail : Bool;
      AlarmCond_BadNoComm1 : Bool;
      AlarmCond_BadNoComm2 : Bool;
      AlarmCond_BadOutOfServ : Bool;
      AlarmCond_BadMaintenance : Bool;
      AlarmCond_BadMaintDemand : Bool;
      AlarmCond_BadNonMeasured : Bool;
      AlarmCond_UncerNonSpec : Bool;
      AlarmCond_UncerLastUseab : Bool;
      AlarmCond_UncerSubstiSet : Bool;
      AlarmCond_UncerIniValue : Bool;
      AlarmCond_UncerSensNotAc : Bool;
      AlarmCond_UncerEUError : Bool;
      AlarmCond_UncerSubNormal : Bool;
      AlarmCond_UncerConfError : Bool;
      AlarmCond_UncerSimValue : Bool;
      AlarmCond_UncerSensCalib : Bool;
      Use_IN_NORM : Bool;   // "1" Use IN_NORM / "0" = Use IN_SCAL
      AlarmCond : Bool;
      FIBUS_SubStatus_Int : Int;
      FIBUS_Quality_Int : Int;
      FIBUS_Limit_Int : Int;
      Raw_Scaled : Real;
      ScaleRange : Real;
      Raw_Normalized : Real;
      DummyReal_1 : Real;
      DummyReal_2 : Real;
      DummyReal_3 : Real;
      AlarmOffLimit : Real;
   END_VAR
   VAR_TEMP   // added for the SCL form of the ladder/FBD networks
      _w1 : Bool;
      _w2 : Bool;
      _w3 : Bool;
      _w4 : Bool;
      _w5 : Bool;
      _w6 : Bool;
      _w7 : Bool;
      _w8 : Bool;
   END_VAR
BEGIN

REGION Network 1: Always On
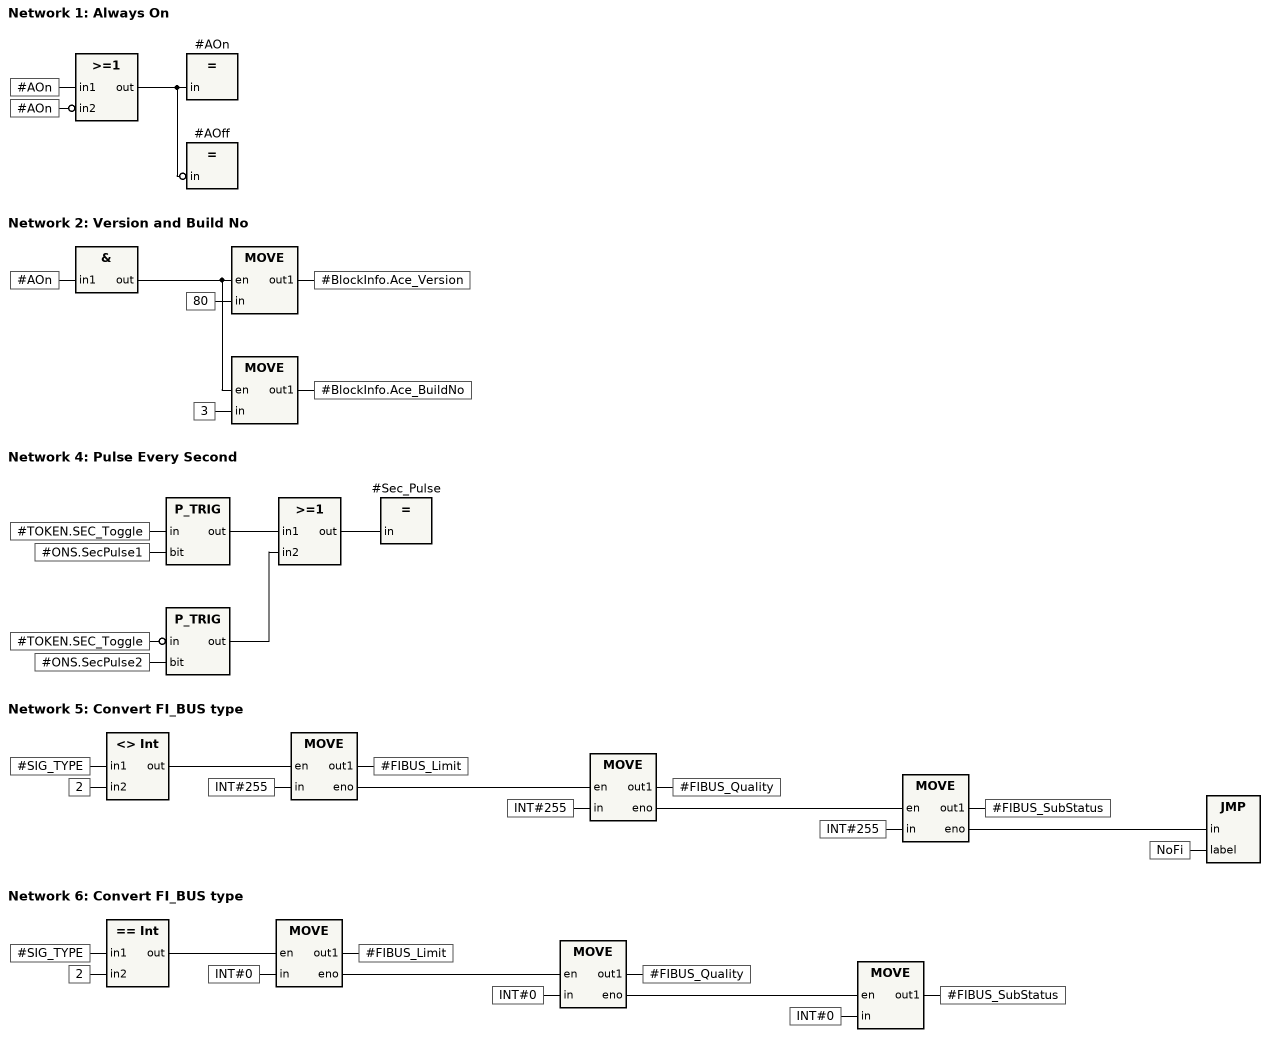
   #AOn := #AOn OR NOT #AOn;
   #AOff := NOT #AOn;
END_REGION

REGION Network 2: Version and Build No
   IF #AOn THEN
       #BlockInfo.Ace_Version := 80;
       #BlockInfo.Ace_BuildNo := 3;
   END_IF;
END_REGION

REGION Network 3 (STL): Instance DB Number to Faceplate
         L     DINO;
         T     #BlockInfo.DB_Number;
END_REGION

REGION Network 4: Pulse Every Second
   #_w1 := #TOKEN.SEC_Toggle AND NOT #ONS.SecPulse1;   // rising edge
   #ONS.SecPulse1 := #TOKEN.SEC_Toggle;
   #_w2 := NOT #TOKEN.SEC_Toggle AND NOT #ONS.SecPulse2;   // rising edge
   #ONS.SecPulse2 := NOT #TOKEN.SEC_Toggle;
   #Sec_Pulse := #_w1 OR #_w2;
END_REGION

REGION Network 5: Convert FI_BUS type
   // ENO of a box is taken as its EN; it also drops when the box reports an error
   #_w1 := #SIG_TYPE <> 2;
   IF #_w1 THEN
       #FIBUS_Limit := INT#255;
       #FIBUS_Quality := INT#255;
       #FIBUS_SubStatus := INT#255;
       GOTO NoFi;
   END_IF;
END_REGION

REGION Network 6: Convert FI_BUS type
   // ENO of a box is taken as its EN; it also drops when the box reports an error
   IF #SIG_TYPE = 2 THEN
       #FIBUS_Limit := INT#0;
       #FIBUS_Quality := INT#0;
       #FIBUS_SubStatus := INT#0;
   END_IF;
END_REGION

REGION Network 7: Convert FI_BUS type
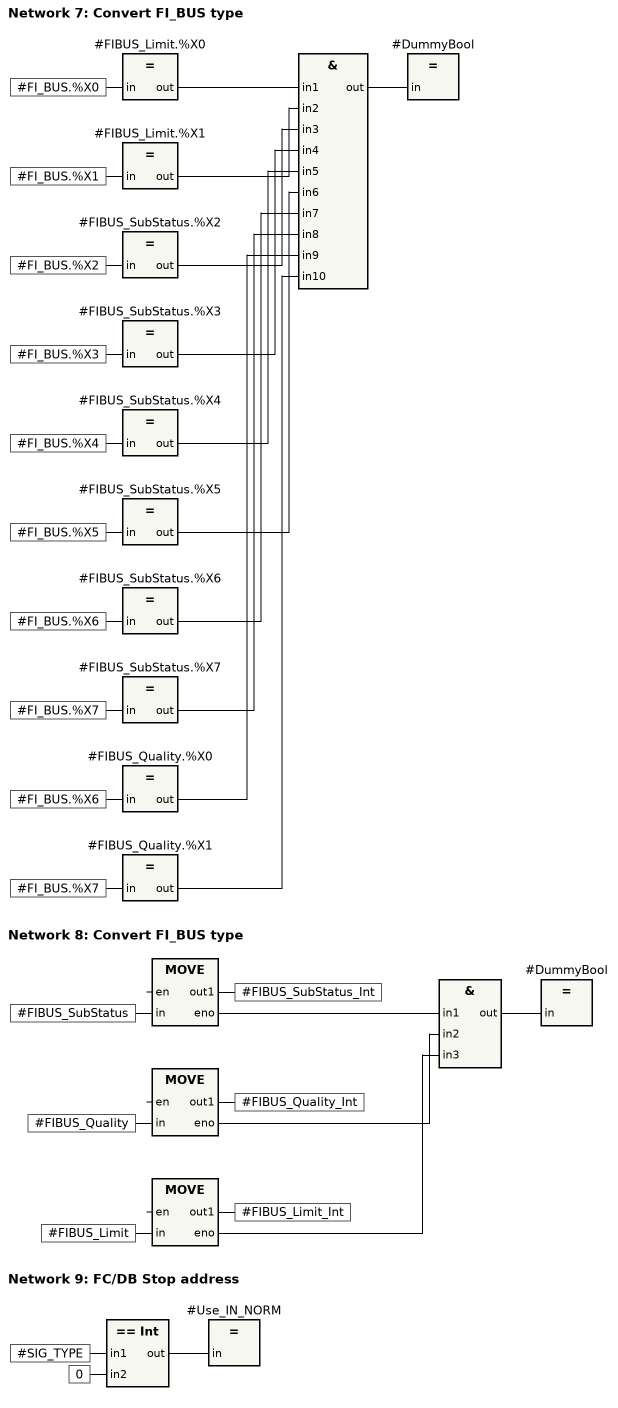
   #FIBUS_Limit.%X0 := #FI_BUS.%X0;
   #FIBUS_Limit.%X1 := #FI_BUS.%X1;
   #FIBUS_SubStatus.%X2 := #FI_BUS.%X2;
   #FIBUS_SubStatus.%X3 := #FI_BUS.%X3;
   #FIBUS_SubStatus.%X4 := #FI_BUS.%X4;
   #FIBUS_SubStatus.%X5 := #FI_BUS.%X5;
   #FIBUS_SubStatus.%X6 := #FI_BUS.%X6;
   #FIBUS_SubStatus.%X7 := #FI_BUS.%X7;
   #FIBUS_Quality.%X0 := #FI_BUS.%X6;
   #FIBUS_Quality.%X1 := #FI_BUS.%X7;
   #DummyBool := #FI_BUS.%X0 AND #FI_BUS.%X1 AND #FI_BUS.%X2 AND #FI_BUS.%X3 AND #FI_BUS.%X4 AND #FI_BUS.%X5 AND #FI_BUS.%X6 AND #FI_BUS.%X7 AND #FI_BUS.%X6 AND #FI_BUS.%X7;
END_REGION

REGION Network 8: Convert FI_BUS type
   NoFi:
   #FIBUS_SubStatus_Int := #FIBUS_SubStatus;
   #FIBUS_Quality_Int := #FIBUS_Quality;
   #FIBUS_Limit_Int := #FIBUS_Limit;
   #DummyBool := TRUE;
END_REGION

REGION Network 9: FC/DB Stop address
   #Use_IN_NORM := #SIG_TYPE = 0;
END_REGION

REGION Network 10: Square / Square Root
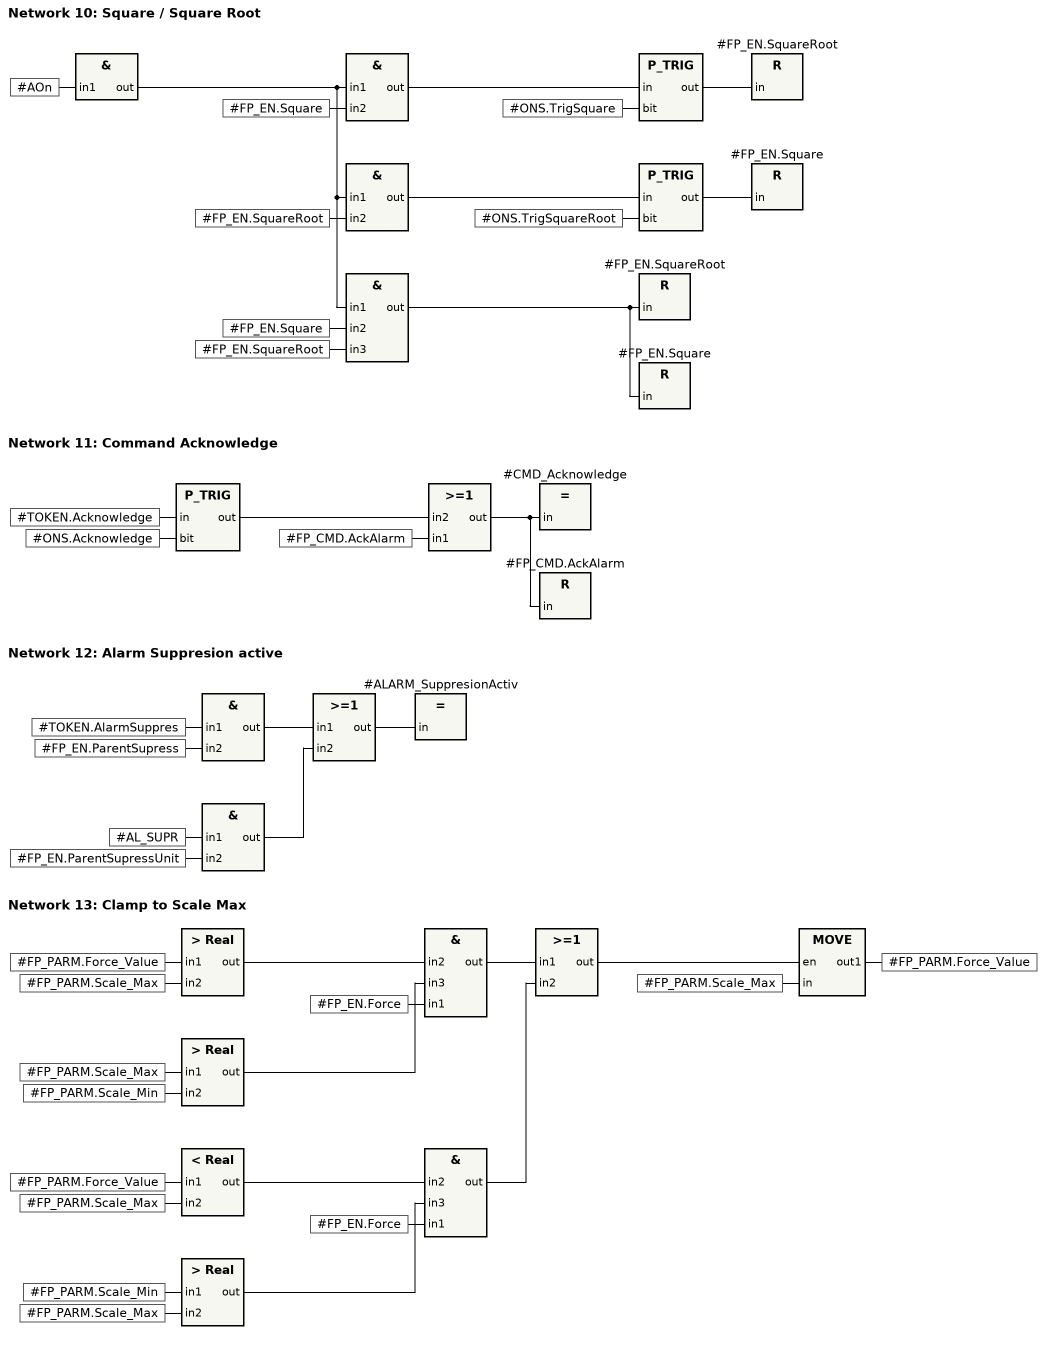
   #_w1 := #AOn AND #FP_EN.Square;
   #_w2 := #_w1 AND NOT #ONS.TrigSquare;   // rising edge
   #ONS.TrigSquare := #_w1;
   IF #_w2 THEN #FP_EN.SquareRoot := FALSE; END_IF;
   #_w3 := #AOn AND #FP_EN.SquareRoot;
   #_w4 := #_w3 AND NOT #ONS.TrigSquareRoot;   // rising edge
   #ONS.TrigSquareRoot := #_w3;
   IF #_w4 THEN #FP_EN.Square := FALSE; END_IF;
   #_w5 := #AOn AND #FP_EN.Square AND #FP_EN.SquareRoot;
   IF #_w5 THEN
       #FP_EN.SquareRoot := FALSE;
       #FP_EN.Square := FALSE;
   END_IF;
END_REGION

REGION Network 11: Command Acknowledge
   // >>>>>>>Automatic Dep_CMD when use of block interface<<<<<<
   #_w1 := #TOKEN.Acknowledge AND NOT #ONS.Acknowledge;   // rising edge
   #ONS.Acknowledge := #TOKEN.Acknowledge;
   #CMD_Acknowledge := #_w1 OR #FP_CMD.AckAlarm;
   IF #CMD_Acknowledge THEN #FP_CMD.AckAlarm := FALSE; END_IF;
END_REGION

REGION Network 12: Alarm Suppresion active
   #ALARM_SuppresionActiv := (#TOKEN.AlarmSuppres AND #FP_EN.ParentSupress) OR (#AL_SUPR AND #FP_EN.ParentSupressUnit);
END_REGION

REGION Network 13: Clamp to Scale Max
   IF ((#FP_PARM.Force_Value > #FP_PARM.Scale_Max) AND (#FP_PARM.Scale_Max > #FP_PARM.Scale_Min) AND #FP_EN.Force) OR ((#FP_PARM.Force_Value < #FP_PARM.Scale_Max) AND (#FP_PARM.Scale_Min > #FP_PARM.Scale_Max) AND #FP_EN.Force) THEN
       #FP_PARM.Force_Value := #FP_PARM.Scale_Max;
   END_IF;
END_REGION

REGION Network 14: Clamp to Scale Min
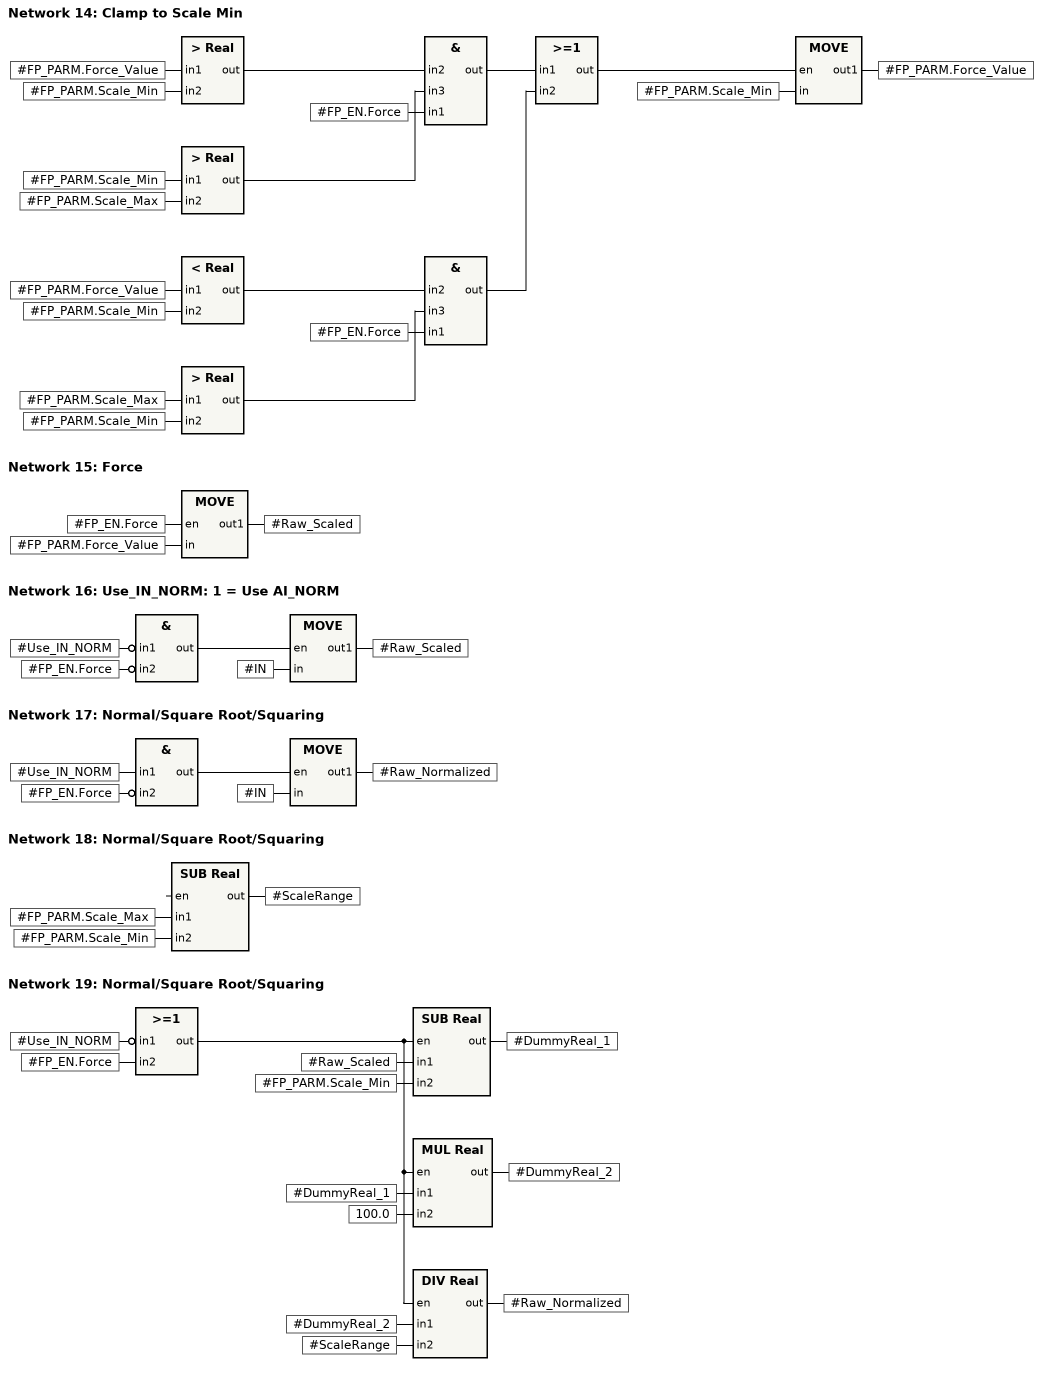
   IF ((#FP_PARM.Force_Value > #FP_PARM.Scale_Min) AND (#FP_PARM.Scale_Min > #FP_PARM.Scale_Max) AND #FP_EN.Force) OR ((#FP_PARM.Force_Value < #FP_PARM.Scale_Min) AND (#FP_PARM.Scale_Max > #FP_PARM.Scale_Min) AND #FP_EN.Force) THEN
       #FP_PARM.Force_Value := #FP_PARM.Scale_Min;
   END_IF;
END_REGION

REGION Network 15: Force
   // >>>>>Force<<<<<
   IF #FP_EN.Force THEN #Raw_Scaled := #FP_PARM.Force_Value; END_IF;
END_REGION

REGION Network 16: Use_IN_NORM: 1 = Use AI_NORM
   IF NOT #Use_IN_NORM AND NOT #FP_EN.Force THEN #Raw_Scaled := #IN; END_IF;
END_REGION

REGION Network 17: Normal/Square Root/Squaring
   IF #Use_IN_NORM AND NOT #FP_EN.Force THEN #Raw_Normalized := #IN; END_IF;
END_REGION

REGION Network 18: Normal/Square Root/Squaring
   #ScaleRange := #FP_PARM.Scale_Max - #FP_PARM.Scale_Min;
END_REGION

REGION Network 19: Normal/Square Root/Squaring
   IF NOT #Use_IN_NORM OR #FP_EN.Force THEN
       #DummyReal_1 := #Raw_Scaled - #FP_PARM.Scale_Min;
       #DummyReal_2 := #DummyReal_1 * 100.0;
       #Raw_Normalized := #DummyReal_2 / #ScaleRange;
   END_IF;
END_REGION

REGION Network 20: Squareroot/Square calculation
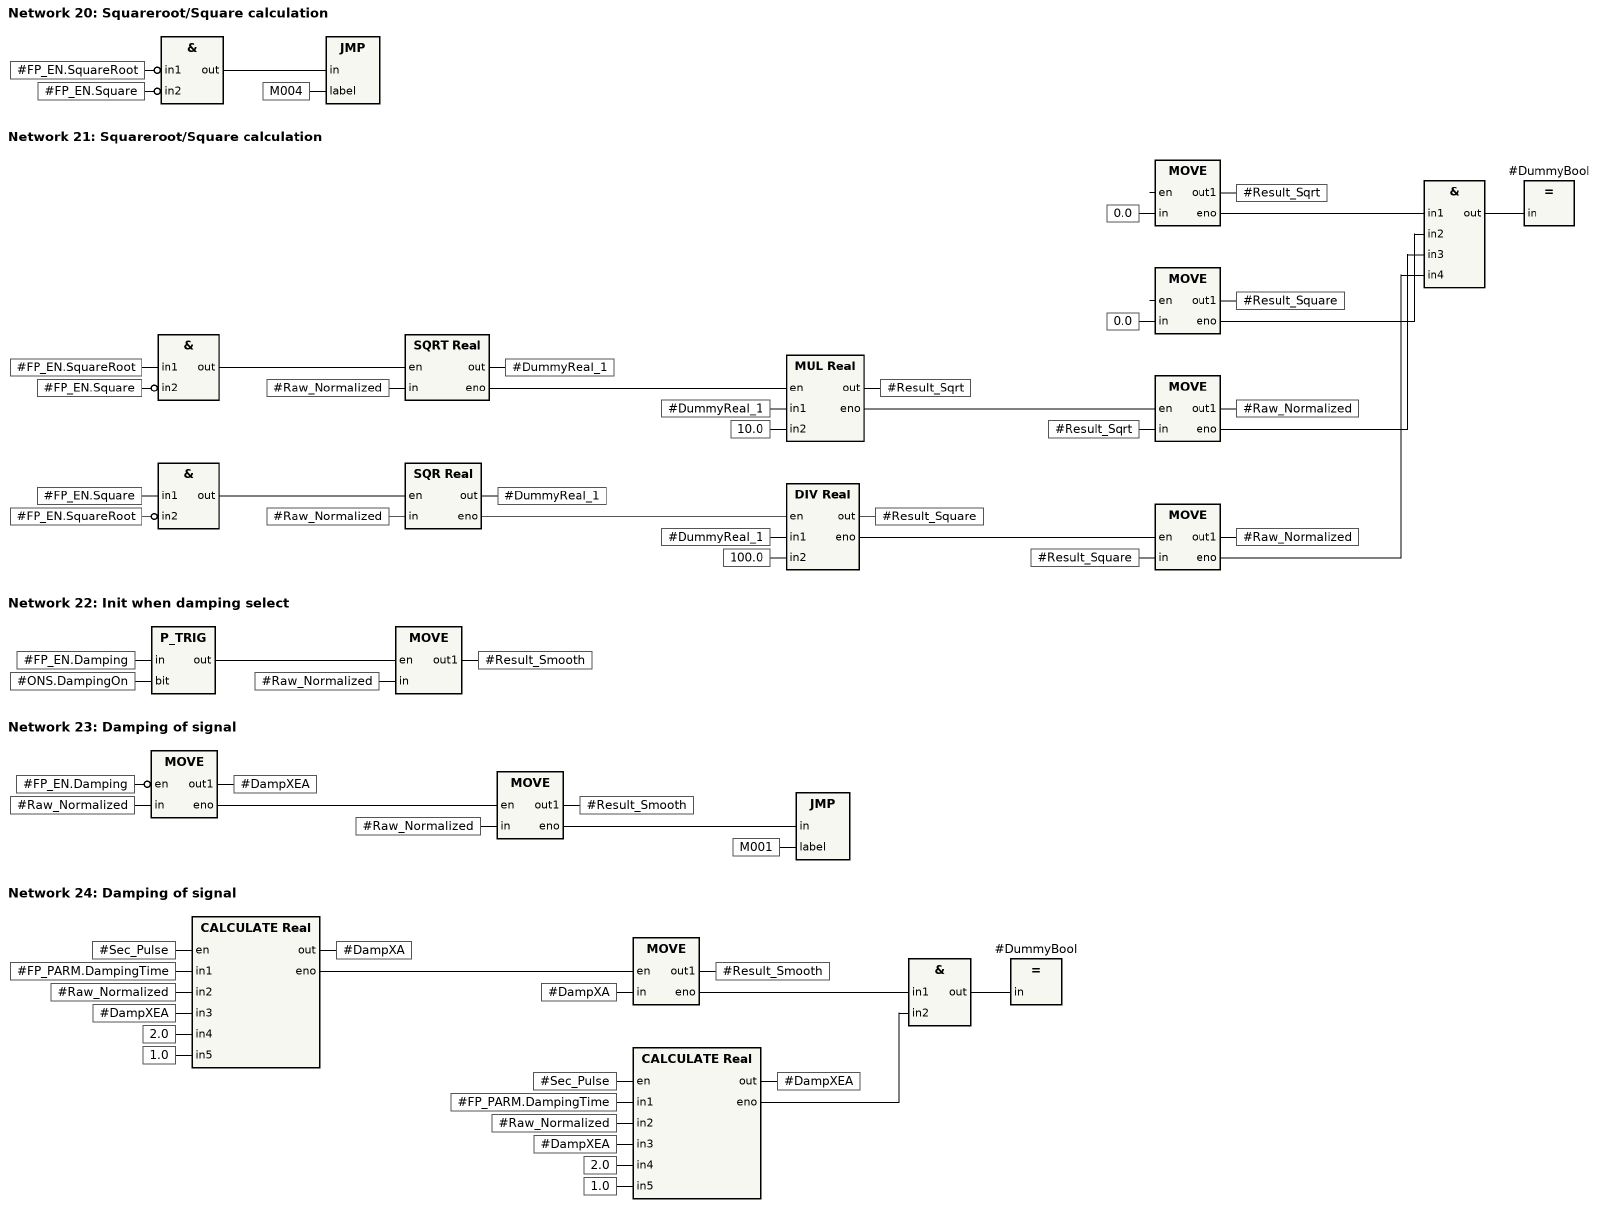
   IF NOT #FP_EN.SquareRoot AND NOT #FP_EN.Square THEN GOTO M004; END_IF;
END_REGION

REGION Network 21: Squareroot/Square calculation
   // ENO of a box is taken as its EN; it also drops when the box reports an error
   #Result_Sqrt := 0.0;
   #Result_Square := 0.0;
   #_w1 := #FP_EN.SquareRoot AND NOT #FP_EN.Square;
   IF #_w1 THEN
       #DummyReal_1 := SQRT(#Raw_Normalized);
       #Result_Sqrt := #DummyReal_1 * 10.0;
       #Raw_Normalized := #Result_Sqrt;
   END_IF;
   #_w2 := #FP_EN.Square AND NOT #FP_EN.SquareRoot;
   IF #_w2 THEN
       #DummyReal_1 := SQR(#Raw_Normalized);
       #Result_Square := #DummyReal_1 / 100.0;
       #Raw_Normalized := #Result_Square;
   END_IF;
   #DummyBool := #_w1 AND #_w2;
END_REGION

REGION Network 22: Init when damping select
   M004:
   #_w1 := #FP_EN.Damping AND NOT #ONS.DampingOn;   // rising edge
   #ONS.DampingOn := #FP_EN.Damping;
   IF #_w1 THEN #Result_Smooth := #Raw_Normalized; END_IF;
END_REGION

REGION Network 23: Damping of signal
   // Damping (smoothing) of signal is based on the trapezoidal formula:
   // XA=(XE-XEA)/1+2TG + XEA  and   XEA=2(XE-XEA)/1+2TG + XEA
   // XE= New analog value
   // XA= Result
   // XEA=Old value for smoothing
   // TG= Damping time
   // TA= Call-up time (allways set to 1 sec.)
   IF NOT #FP_EN.Damping THEN
       #DampXEA := #Raw_Normalized;
       #Result_Smooth := #Raw_Normalized;
       GOTO M001;
   END_IF;
END_REGION

REGION Network 24: Damping of signal
   // Damping (smoothing) of signal is based on the trapezoidal formula:
   // XA=(XE-XEA)/1+2TG + XEA  and   XEA=2(XE-XEA)/1+2TG + XEA
   // XE= New analog value
   // XA= Result
   // XEA=Old value for smoothing
   // TG= Damping time
   // TA= Call-up time (allways set to 1 sec.)
   IF #Sec_Pulse THEN
       #DampXA := (#DampXEA + ((#Raw_Normalized-#DampXEA) / ((#FP_PARM.DampingTime * 2.0) + 1.0)));
       #Result_Smooth := #DampXA;
       #DampXEA := (#DampXEA + (((#Raw_Normalized-#DampXEA)*2.0) / ((#FP_PARM.DampingTime * 2.0) + 1.0)));
   END_IF;
   #DummyBool := #Sec_Pulse AND #Sec_Pulse;
END_REGION

REGION Network 25: Signal limit calculation
   // Descide source for analog value
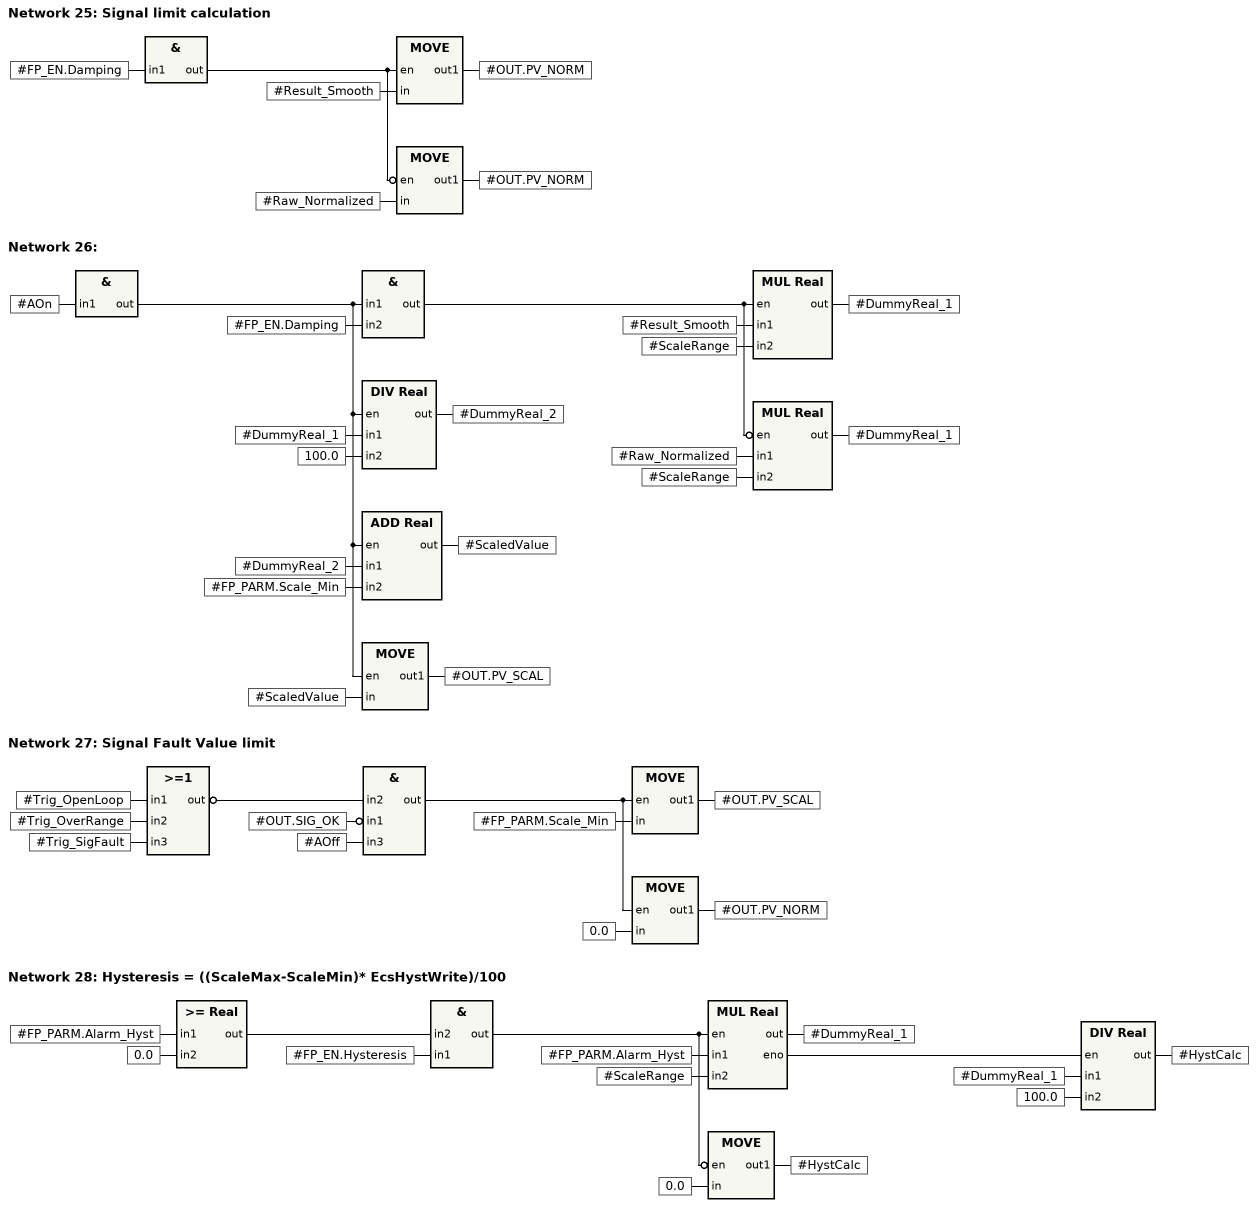
   M001:
   IF #FP_EN.Damping THEN #OUT.PV_NORM := #Result_Smooth; END_IF;
   IF NOT #FP_EN.Damping THEN #OUT.PV_NORM := #Raw_Normalized; END_IF;
END_REGION

REGION Network 26
   // >>>>>Scaling Analog Input<<<<<
   #_w1 := #AOn AND #FP_EN.Damping;
   IF #_w1 THEN #DummyReal_1 := #Result_Smooth * #ScaleRange; END_IF;
   IF NOT #_w1 THEN #DummyReal_1 := #Raw_Normalized * #ScaleRange; END_IF;
   IF #AOn THEN
       #DummyReal_2 := #DummyReal_1 / 100.0;
       #ScaledValue := #DummyReal_2 + #FP_PARM.Scale_Min;
       #OUT.PV_SCAL := #ScaledValue;
   END_IF;
END_REGION

REGION Network 27: Signal Fault Value limit
   // Build 002 - 26 March 2019 : The network is not allowed to execute, therby the PV_SCAl & PV_NORM shall be scaled linearly to the input signal with reference to Scale Min/Max
   IF NOT (#Trig_OpenLoop OR #Trig_OverRange OR #Trig_SigFault) AND NOT #OUT.SIG_OK AND #AOff THEN
       #OUT.PV_SCAL := #FP_PARM.Scale_Min;
       #OUT.PV_NORM := 0.0;
   END_IF;
END_REGION

REGION Network 28: Hysteresis = ((ScaleMax-ScaleMin)* EcsHystWrite)/100
   // >>>>>Calculate Hysteresis Value<<<<<
   // ENO of a box is taken as its EN; it also drops when the box reports an error
   #_w1 := (#FP_PARM.Alarm_Hyst >= 0.0) AND #FP_EN.Hysteresis;
   IF #_w1 THEN
       #DummyReal_1 := #FP_PARM.Alarm_Hyst * #ScaleRange;
       #HystCalc := #DummyReal_1 / 100.0;
   END_IF;
   IF NOT #_w1 THEN #HystCalc := 0.0; END_IF;
END_REGION

REGION Network 29: Open Loop Delay
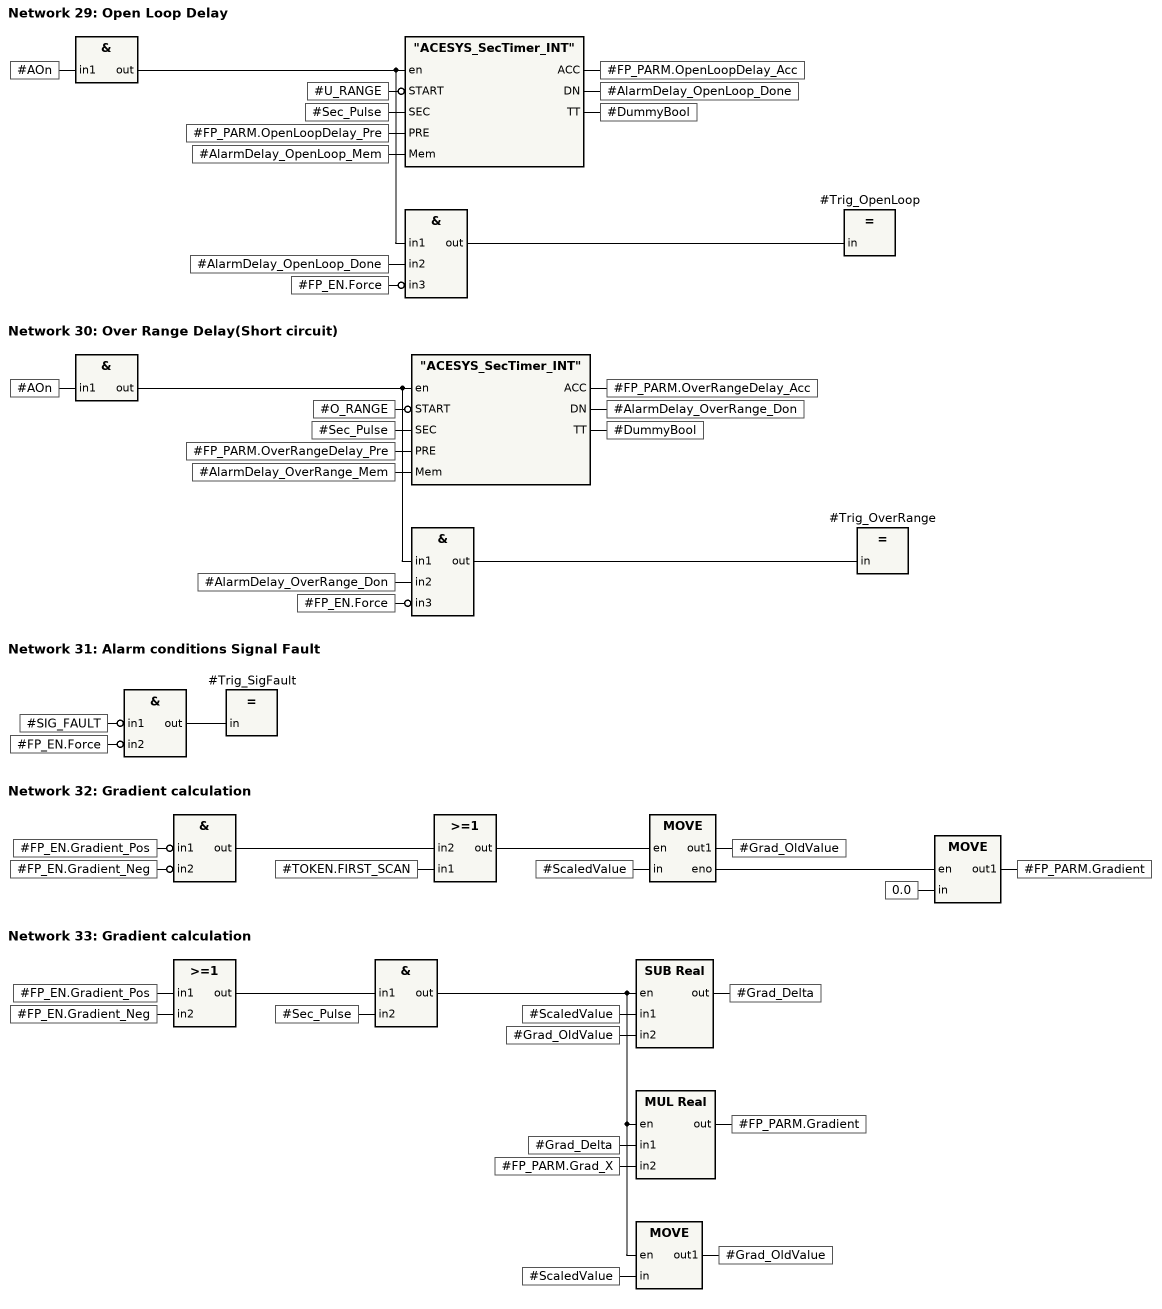
   IF #AOn THEN
       "ACESYS_SecTimer_INT"(START := NOT #U_RANGE,
                             SEC := #Sec_Pulse,
                             PRE := #FP_PARM.OpenLoopDelay_Pre,
                             Mem := #AlarmDelay_OpenLoop_Mem,
                             ACC => #FP_PARM.OpenLoopDelay_Acc,
                             DN => #AlarmDelay_OpenLoop_Done,
                             TT => #DummyBool);
   END_IF;
   #Trig_OpenLoop := #AOn AND #AlarmDelay_OpenLoop_Done AND NOT #FP_EN.Force;
END_REGION

REGION Network 30: Over Range Delay(Short circuit)
   IF #AOn THEN
       "ACESYS_SecTimer_INT"(START := NOT #O_RANGE,
                             SEC := #Sec_Pulse,
                             PRE := #FP_PARM.OverRangeDelay_Pre,
                             Mem := #AlarmDelay_OverRange_Mem,
                             ACC => #FP_PARM.OverRangeDelay_Acc,
                             DN => #AlarmDelay_OverRange_Don,
                             TT => #DummyBool);
   END_IF;
   #Trig_OverRange := #AOn AND #AlarmDelay_OverRange_Don AND NOT #FP_EN.Force;
END_REGION

REGION Network 31: Alarm conditions Signal Fault
   // >>>>>Signal Fault<<<<<
   #Trig_SigFault := NOT #SIG_FAULT AND NOT #FP_EN.Force;
END_REGION

REGION Network 32: Gradient calculation
   // >>>>>Gradient calculation<<<<<
   // 
   // The differentiation signal is calculated by:
   // dY/dT=(New processvalue - Old processvalue) * X-factor.
   // The X-factor is used to magnify the value.
   // ENO of a box is taken as its EN; it also drops when the box reports an error
   IF (NOT #FP_EN.Gradient_Pos AND NOT #FP_EN.Gradient_Neg) OR #TOKEN.FIRST_SCAN THEN
       #Grad_OldValue := #ScaledValue;
       #FP_PARM.Gradient := 0.0;
   END_IF;
END_REGION

REGION Network 33: Gradient calculation
   IF (#FP_EN.Gradient_Pos OR #FP_EN.Gradient_Neg) AND #Sec_Pulse THEN
       #Grad_Delta := #ScaledValue - #Grad_OldValue;
       #FP_PARM.Gradient := #Grad_Delta * #FP_PARM.Grad_X;
       #Grad_OldValue := #ScaledValue;
   END_IF;
END_REGION

REGION Network 34: Gradient Condition
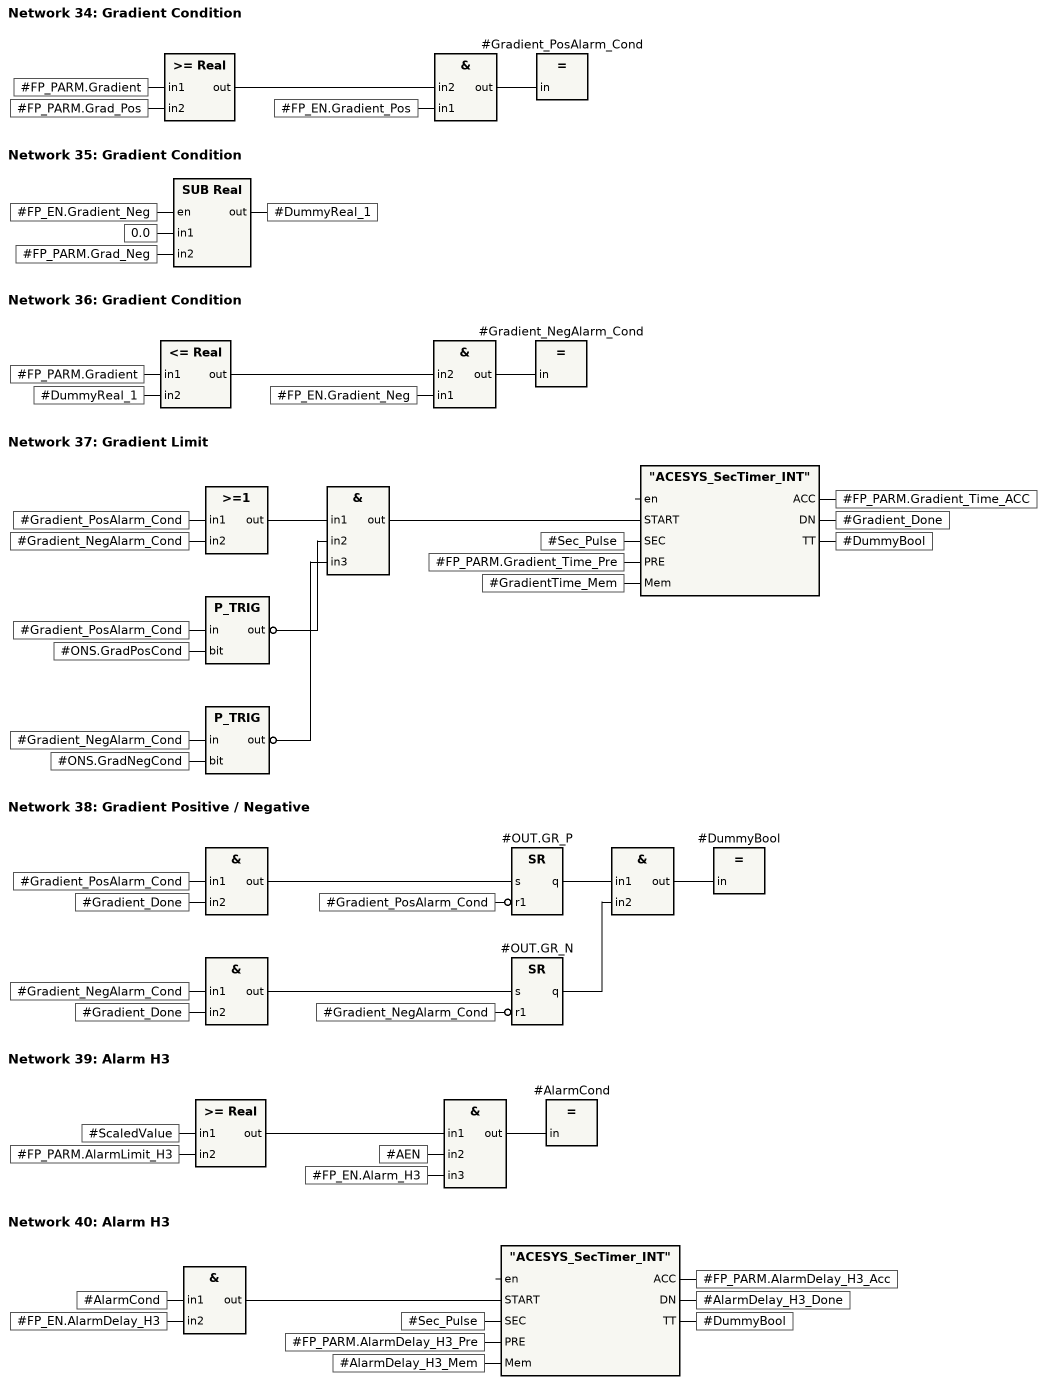
   #Gradient_PosAlarm_Cond := (#FP_PARM.Gradient >= #FP_PARM.Grad_Pos) AND #FP_EN.Gradient_Pos;
END_REGION

REGION Network 35: Gradient Condition
   IF #FP_EN.Gradient_Neg THEN #DummyReal_1 := 0.0 - #FP_PARM.Grad_Neg; END_IF;
END_REGION

REGION Network 36: Gradient Condition
   #Gradient_NegAlarm_Cond := (#FP_PARM.Gradient <= #DummyReal_1) AND #FP_EN.Gradient_Neg;
END_REGION

REGION Network 37: Gradient Limit
   // Announciation limits for gradient and announciation delay.
   #_w1 := #Gradient_PosAlarm_Cond AND NOT #ONS.GradPosCond;   // rising edge
   #ONS.GradPosCond := #Gradient_PosAlarm_Cond;
   #_w2 := #Gradient_NegAlarm_Cond AND NOT #ONS.GradNegCond;   // rising edge
   #ONS.GradNegCond := #Gradient_NegAlarm_Cond;
   "ACESYS_SecTimer_INT"(START := (#Gradient_PosAlarm_Cond OR #Gradient_NegAlarm_Cond) AND NOT #_w1 AND NOT #_w2,
                         SEC := #Sec_Pulse,
                         PRE := #FP_PARM.Gradient_Time_Pre,
                         Mem := #GradientTime_Mem,
                         ACC => #FP_PARM.Gradient_Time_ACC,
                         DN => #Gradient_Done,
                         TT => #DummyBool);
END_REGION

REGION Network 38: Gradient Positive / Negative
   IF #Gradient_PosAlarm_Cond AND #Gradient_Done THEN
       #OUT.GR_P := TRUE;   // SR flip-flop
   END_IF;
   IF NOT #Gradient_PosAlarm_Cond THEN #OUT.GR_P := FALSE; END_IF;
   IF #Gradient_NegAlarm_Cond AND #Gradient_Done THEN
       #OUT.GR_N := TRUE;   // SR flip-flop
   END_IF;
   IF NOT #Gradient_NegAlarm_Cond THEN #OUT.GR_N := FALSE; END_IF;
   #DummyBool := #OUT.GR_P AND #OUT.GR_N;
END_REGION

REGION Network 39: Alarm H3
   #AlarmCond := (#ScaledValue >= #FP_PARM.AlarmLimit_H3) AND #AEN AND #FP_EN.Alarm_H3;
END_REGION

REGION Network 40: Alarm H3
   "ACESYS_SecTimer_INT"(START := #AlarmCond AND #FP_EN.AlarmDelay_H3,
                         SEC := #Sec_Pulse,
                         PRE := #FP_PARM.AlarmDelay_H3_Pre,
                         Mem := #AlarmDelay_H3_Mem,
                         ACC => #FP_PARM.AlarmDelay_H3_Acc,
                         DN => #AlarmDelay_H3_Done,
                         TT => #DummyBool);
END_REGION

REGION Network 41: H3 // Alarm conditions H3
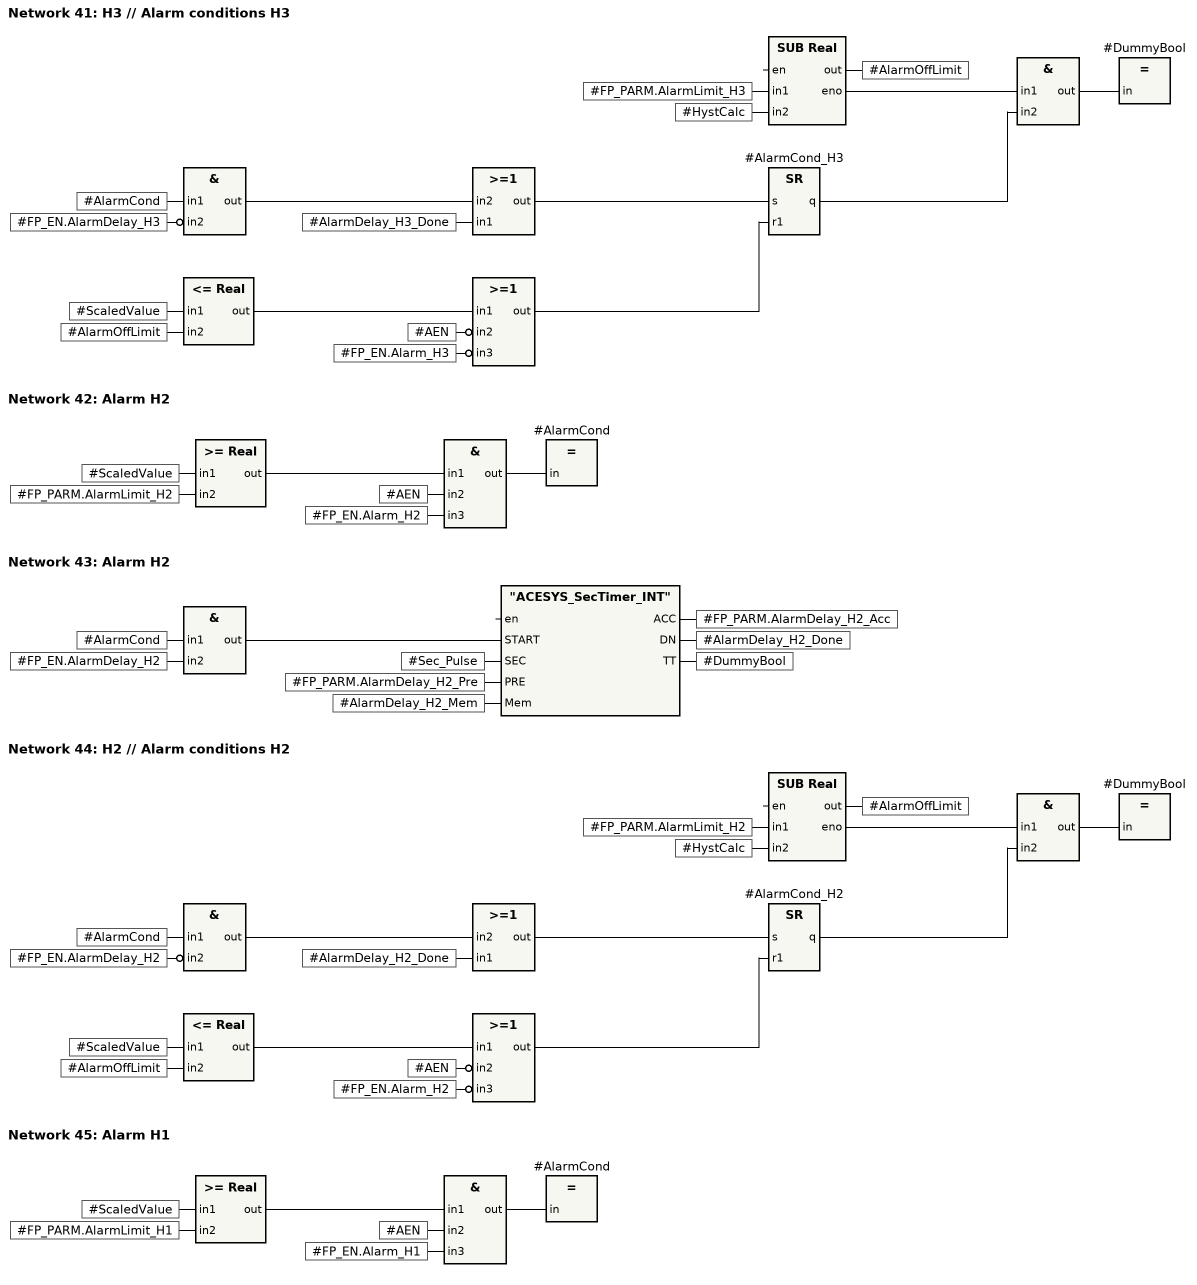
   // ENO of a box is taken as its EN; it also drops when the box reports an error
   #AlarmOffLimit := #FP_PARM.AlarmLimit_H3 - #HystCalc;
   IF (#AlarmCond AND NOT #FP_EN.AlarmDelay_H3) OR #AlarmDelay_H3_Done THEN
       #AlarmCond_H3 := TRUE;   // SR flip-flop
   END_IF;
   IF (#ScaledValue <= #AlarmOffLimit) OR NOT #AEN OR NOT #FP_EN.Alarm_H3 THEN
       #AlarmCond_H3 := FALSE;
   END_IF;
   #DummyBool := #AlarmCond_H3;
END_REGION

REGION Network 42: Alarm H2
   #AlarmCond := (#ScaledValue >= #FP_PARM.AlarmLimit_H2) AND #AEN AND #FP_EN.Alarm_H2;
END_REGION

REGION Network 43: Alarm H2
   "ACESYS_SecTimer_INT"(START := #AlarmCond AND #FP_EN.AlarmDelay_H2,
                         SEC := #Sec_Pulse,
                         PRE := #FP_PARM.AlarmDelay_H2_Pre,
                         Mem := #AlarmDelay_H2_Mem,
                         ACC => #FP_PARM.AlarmDelay_H2_Acc,
                         DN => #AlarmDelay_H2_Done,
                         TT => #DummyBool);
END_REGION

REGION Network 44: H2 // Alarm conditions H2
   // ENO of a box is taken as its EN; it also drops when the box reports an error
   #AlarmOffLimit := #FP_PARM.AlarmLimit_H2 - #HystCalc;
   IF (#AlarmCond AND NOT #FP_EN.AlarmDelay_H2) OR #AlarmDelay_H2_Done THEN
       #AlarmCond_H2 := TRUE;   // SR flip-flop
   END_IF;
   IF (#ScaledValue <= #AlarmOffLimit) OR NOT #AEN OR NOT #FP_EN.Alarm_H2 THEN
       #AlarmCond_H2 := FALSE;
   END_IF;
   #DummyBool := #AlarmCond_H2;
END_REGION

REGION Network 45: Alarm H1
   #AlarmCond := (#ScaledValue >= #FP_PARM.AlarmLimit_H1) AND #AEN AND #FP_EN.Alarm_H1;
END_REGION

REGION Network 46: Alarm H1
